	Original Author(s): Rob Remillard of Sodecia GTAC.; 
------------------------------------------------------------------------------------------
REVISION NOTES:
	Version 20150203
		- intial concept, r.remillard
	Version 20151105
		- added discrete_image to var_output to expose for visualization on UIs, b.lekx-toniolo
		- added Not Comm_Error interlock to Locked and Unlocked Signals for redundancy, b.lekx-toniolo
------------------------------------------------------------------------------------------
*)



FUNCTION_BLOCK FB_ATI_Changer_20151105

VAR_INPUT

	ATI_Lock_Requested:				BOOL;
	ATI_Unlock_Requested:			BOOL;
	Fault_Reset:						BOOL;

END_VAR

VAR

	In_From_Hardware AT %I*: 			udt_ATI_Input_20150203;
	Out_To_Hardware AT %Q*:			udt_ATI_Output_20150203;

	Lock_ATI:						BOOL;
	Unlock_ATI:						BOOL;

	(*Input Signals From ATI*)
	US1_Power_Present:				BOOL;
	US2_Power_Present:				BOOL;
	RTL1:							BOOL;
	RTL2:							BOOL;
	Tool_Present:					BOOL;
	Tool_PWR_Present:				BOOL;

	TSIV:							BOOL;
	TSRV:							BOOL;
	RTLV1:							BOOL;
	RTLV2:							BOOL;

	Tool_ID:							UDINT;

	Error_On_Lock:					BOOL;
	Error_On_Unlock:					BOOL;


	DiscreteNode_OK: 				BOOL;
	ECatSlave_Cable_Breaks:			UDINT;

END_VAR

VAR_OUTPUT

	FB_OK:							BOOL;
	Discrete_Image:					udt_ATIxx_Image_20151104;
	ATI_Sensors_On:					BOOL;
	ATI_Locked:						BOOL;
	ATI_Unlocked:					BOOL;
	ATI_Unlock_Enabled:				BOOL;
	Tool_ID_Out0:					BOOL;
	Tool_ID_Out1:					BOOL;
	Tool_ID_Out2:					BOOL;
	Tool_ID_Out3:					BOOL;
	Tool_ID_Out4:					BOOL;
	Tool_ID_Out5:					BOOL;
	Tool_ID_Out6:					BOOL;
	Tool_ID_Out7:					BOOL;
	Unsafe_Unlock:					BOOL;
	Sensor_Fault:						BOOL;
	COMM_Error:						BOOL;

END_VAR

	(*Set FB_OK to True*)
	FB_OK:= TRUE;

(*$$$$$$$$$$$$$$$$$$$$$$$$$$$$$$$$$$$$$$$$$$$$$$$$Gather Status Of Hardware $$$$$$$$$$$$$$$$$$$$$$$$$$$$$$$$$$$$$$$$$$$$$$$$$$$$*)
	(*Discrete I/O Nodes*)
	IF In_From_Hardware.InfoData.State=8

		THEN
			DiscreteNode_OK:=TRUE;

	ELSE
			DiscreteNode_OK:=FALSE;

	END_IF;


	(*Cable Break Detection*)
	ECatSlave_Cable_Breaks:= FUN_GTAC_EcatSlaveConnState
							(In_From_Hardware.InfoData.State,
							0,0,0,0,0,0,0,0,0,0,0,0,0,0,0,0,0,0,0,0,0,0,0,0,0,0,0,0,0); (*Function Returns Flags to warn of possible cable break*)

(*----------------------------------------------------------------------------------------------------------------------------------------------------------------------------------------------------------*)

(*+++++++++++++++++++++++++++Input Byte Mapping+++++++++++++++++++++++++++*)

	ATI_Locked:= In_From_Hardware.Byte0.0 AND NOT Comm_Error;				(*ATI Locked Status from VL1*)
	ATI_Unlocked:= In_From_Hardware.Byte0.1 AND NOT Comm_Error;				(*ATI Unlocked Status from VL1*)
	US1_Power_Present:= In_From_Hardware.Byte0.2;								(*ATI Main Power Present*)
	US2_Power_Present:= In_From_Hardware.Byte0.3;								(*ATI Valve Power Present*)
	RTL1:= In_From_Hardware.Byte0.4;											(*ATI Ready To Lock Prox 1*)
	RTL2:= In_From_Hardware.Byte0.5;											(*ATI Ready To Lock Prox 2*)
	Tool_Present:= In_From_Hardware.Byte0.6;									(*ATI Master and Tool are in Electrical Contact*)
	Tool_PWR_Present:= In_From_Hardware.Byte0.7;								(*ATI Arc Prevention Circuit on and power to Tool*)

	ATI_Unlock_Enabled:= In_From_Hardware.Byte1.0;								(*ATI Unlock Enabled*)
	TSIV:= In_From_Hardware.Byte1.1;											(*ATI Tool Stand Interlock Switch Verify*)
	TSRV:= In_From_Hardware.Byte1.2;											(*ATI Tool Stand Interlock Relay Verify*)
	RTLV1:= In_From_Hardware.Byte1.4;											(*ATI Ready To Lock Relay1 Verify*)
	RTLV2:= In_From_Hardware.Byte1.5;											(*ATI Ready To Lock Relay2 Verify*)

	Error_On_Lock:= In_From_Hardware.Byte2.0;									(*ATI Overload or Short Circuit on Latch Output*)
	Error_On_Unlock:= In_From_Hardware.Byte2.1;									(*ATI Overload or Short Circuit on Unlatch Output*)
	Unsafe_Unlock:= In_From_Hardware.Byte2.3;									(*ATI Unlatch rejected due to unsafe condition present*)
	Sensor_Fault:= In_From_Hardware.Byte2.4;									(*ATI Lock and Unlock inputs true at the same time*)
	COMM_Error:= In_From_Hardware.Byte2.5;									(*ATI Tool ID Communication Timeout*)

	Tool_ID:=  In_From_Hardware.Byte456;										(*ATI Tool ID*)

	Tool_ID_Out0:= Tool_ID.0;
	Tool_ID_Out1:= Tool_ID.1;
	Tool_ID_Out2:= Tool_ID.2;
	Tool_ID_Out3:= Tool_ID.3;
	Tool_ID_Out4:= Tool_ID.4;
	Tool_ID_Out5:= Tool_ID.5;
	Tool_ID_Out6:= Tool_ID.6;
	Tool_ID_Out7:= Tool_ID.7;



(*+++++++++++++++++++++++++++++ATI Control Code++++++++++++++++++++++++++++*)

	IF ATI_Lock_Requested
		THEN
			Lock_ATI:= TRUE;
			Unlock_ATI:= FALSE;
	ELSIF NOT Tool_Present AND NOT ATI_Lock_Requested
		THEN
			Lock_ATI:= FALSE;
	END_IF;

	IF ATI_Unlock_Requested AND TSIV AND TSRV AND ATI_Unlock_Enabled
		THEN
			Lock_ATI:= FALSE;
			Unlock_ATI:= NOT Lock_ATI;
	END_IF;

	ATI_Sensors_On:= RTL1 AND RTL2;

(*$$$$$$$$$$$$$$$$$$$$$$$$$$$$$$$$$$$$$$$$$$$$$$ Transfer Standard Outputs $$$$$$$$$$$$$$$$$$$$$$$$$$$$$$$$$$$$$$$$$$$*)
	(*Transfer I/O Images for Display On UI*)
Discrete_Image.In_From_Hardware:= In_From_Hardware;
Discrete_Image.Out_To_Hardware:= Out_To_Hardware;
Discrete_Image.ECatSlave_Cable_Breaks:= ECatSlave_Cable_Breaks;

(*+++++++++++++++++++++++++++Output Byte Mapping+++++++++++++++++++++++++++*)

	Out_To_Hardware.Byte0.0:= Lock_ATI;					(*Request Lock*)
	Out_To_Hardware.Byte0.1:= Unlock_ATI;					(*Request Unlock*)
	Out_To_Hardware.Byte0.3:= Fault_Reset;					(*Reset Errors, allow affected I/O to be reactivated*)

END_FUNCTION_BLOCK

// ---- POUs/FBs/FB_GTAC_WaterStand_20220622.TcPOU
(*FB to handle robot water tower
	Version: 20170801
	- combined FB_GTAC_Robot_TempFlow and FB_GTAC_Fixture_Single into one FB, j.vandongen
	- added option to choose between 1 output and 2 output (in the case of a fixture where only one is required), j.vandongen
	Version 20171111
	- changed Timeout reset to rising edge trigger, j.vandongen 
	- added var out for coolig ok, j.vandongen
	Version 20190726
	- added outputs for the control of the water saver unit, j.vandongen
	Version 20200710
	- removed cards EP3174 and EP2028. changed to EP6224 IO-Link, j.vandongen
	Version 20200917
	- corrected error in fault code for DegreesC2, j.vandongen
	Version 20201125
	- corrected mapping issue causing incorrect flow to be shown, j.vandongen
	Version 20220131
	- added mapping for using the inport ports in the I/O Link cards, j. underhill
	Version 20220622
	- fixes for issues found with negative flow values (see 5.06 GH issues #2 notes), b.lekx-toniolo, j.underhill, d.esteves, c.drees
		NOTE: (from brent) the issue is we take a signed value from the meter and shove it into a UINT bit by bit....I'm not sure why the original developer did this but it should be re-examined as a whole


*)

FUNCTION_BLOCK FB_GTAC_WaterStand_20220622

VAR_INPUT

	Enable_Timeout: BOOL; 	(*Enable Timeout to shut off valve if flow not achieved in time*)
	Timeout_Reset: BOOL;		(*Reset (Retry) Timepout*)
	Timeout_SetPoint: TIME;	(*TimeoutSetpoint Input, limited to 1-10S*)

	TempHighLimit1: REAL;
	TempHighLimit2: REAL;
	FlowLowLimit1: REAL;
	FlowLowLimit2: REAL;

	Option_WaterCount: INT;

	Valve1: BOOL;
	Valve2: BOOL;
	Valve3: BOOL;
	Valve4: BOOL;


END_VAR

VAR

(*Hardware Related Data Types*)
	(*Develop "Beckhoff Nodes"*)
	N01 AT %I*: udt_EP6224;
	N01_I AT %I*: udt_EP6224_I;
	N01_CMD AT %Q*: udt_EP6224_CMD;

(* Nodes States*)
	DiscreteNode_OK: BOOL;

(*Cable Break States*)
	ECatSlave_Cable_Breaks: UDINT;

	Fault_Tmrs: ARRAY [0..10] OF TON;
	Temperature1_Fault_Delay_TMR : BOOL;
	Temperature2_Fault_Delay_TMR : BOOL;
	Flow1_Fault_Delay_TMR : BOOL;
	Flow2_Fault_Delay_TMR : BOOL;

	RawTemp1: UINT;
	RawTemp2: UINT;

	RawFlow1: UINT;
	RawFlow2: UINT;

	TempReal1: REAL;
	TempReal2: REAL;
	FlowReal1: REAL;
	FlowReal2: REAL;

	DegreesC1: REAL;
	DegreesC2: REAL;

	Flow_lpm1: REAL;
	Flow_lpm2: REAL;

	WaterTempFlow_OK: BOOL;

	Reset_Req: R_TRIG;


END_VAR

VAR_OUTPUT

	Discrete_Image: udt_WaterStand_Image_20220131;

	Temperature_Fault1: BOOL;
	Temperature_Fault2: BOOL;
	Flow_Fault1: BOOL;
	Flow_Fault2: BOOL;

	Cooling_OK: BOOL;

END_VAR

(*$$$$$$$$$$$$$$$$$$$$$$$$$$$$$$$$$$$$$$$$$$$$$$$$Gather Status Of Hardware $$$$$$$$$$$$$$$$$$$$$$$$$$$$$$$$$$$$$$$$$$$$$$$$$$$$*)
	(*Discrete I/O Nodes*)
	IF (N01.InfoData.State=8)

		THEN DiscreteNode_OK:=TRUE;
	ELSE DiscreteNode_OK:=FALSE;
	END_IF;
	(*Cable Break Detection*)
	ECatSlave_Cable_Breaks:= FUN_GTAC_EcatSlaveConnState
							(N01.InfoData.State,
							0,0,0,0,0,0,0,0,0,0,0,0,0,0,0,0,0,0,0,0,0,0,0,0,0,0,0,0,0); (*Function Returns Flags to warn of possible cable break*)




(*----------------------------------------------------Temperature conversion and output----------------------------------------------------*)
	RawTemp1.0:= N01.Port1_ProcessData[7].2;
	RawTemp1.1:= N01.Port1_ProcessData[7].3;
	RawTemp1.2:= N01.Port1_ProcessData[7].4;
	RawTemp1.3:= N01.Port1_ProcessData[7].5;
	RawTemp1.4:= N01.Port1_ProcessData[7].6;
	RawTemp1.5:= N01.Port1_ProcessData[7].7;
	RawTemp1.6:= N01.Port1_ProcessData[6].0;
	RawTemp1.7:= N01.Port1_ProcessData[6].1;
	RawTemp1.8:= N01.Port1_ProcessData[6].2;
	RawTemp1.9:= N01.Port1_ProcessData[6].3;
	RawTemp1.10:= N01.Port1_ProcessData[6].4;
	RawTemp1.11:= N01.Port1_ProcessData[6].5;
	RawTemp1.12:= N01.Port1_ProcessData[6].6;
	RawTemp1.13:= N01.Port1_ProcessData[6].7;

	TempReal1:= RawTemp1 * 0.1; (*gradient to shift decimal place*)

	RawTemp2.0:= N01.Port2_ProcessData[7].2;
	RawTemp2.1:= N01.Port2_ProcessData[7].3;
	RawTemp2.2:= N01.Port2_ProcessData[7].4;
	RawTemp2.3:= N01.Port2_ProcessData[7].5;
	RawTemp2.4:= N01.Port2_ProcessData[7].6;
	RawTemp2.5:= N01.Port2_ProcessData[7].7;
	RawTemp2.6:= N01.Port2_ProcessData[6].0;
	RawTemp2.7:= N01.Port2_ProcessData[6].1;
	RawTemp2.8:= N01.Port2_ProcessData[6].2;
	RawTemp2.9:= N01.Port2_ProcessData[6].3;
	RawTemp2.10:= N01.Port2_ProcessData[6].4;
	RawTemp2.11:= N01.Port2_ProcessData[6].5;
	RawTemp2.12:= N01.Port2_ProcessData[6].6;
	RawTemp2.13:= N01.Port2_ProcessData[6].7;

	TempReal2:= RawTemp2 * 0.1; (*gradient to shift decimal place*)

(*Set the scale of the input value to match the temperature switch*)
	DegreesC1:= TempReal1;			(*Scale value determined at setup*)
	DegreesC2:= TempReal2;			(*Scale value determined at setup*)



(*----------------------------------------------------------Flow conversion and Output-------------------------------------------------------*)
	RawFlow1.0:= N01.Port1_ProcessData[5].0;
	RawFlow1.1:= N01.Port1_ProcessData[5].1;
	RawFlow1.2:= N01.Port1_ProcessData[5].2;
	RawFlow1.3:= N01.Port1_ProcessData[5].3;
	RawFlow1.4:= N01.Port1_ProcessData[5].4;
	RawFlow1.5:= N01.Port1_ProcessData[5].5;
	RawFlow1.6:= N01.Port1_ProcessData[5].6;
	RawFlow1.7:= N01.Port1_ProcessData[5].7;
	RawFlow1.8:= N01.Port1_ProcessData[4].0;
	RawFlow1.9:= N01.Port1_ProcessData[4].1;
	RawFlow1.10:= N01.Port1_ProcessData[4].2;
	RawFlow1.11:= N01.Port1_ProcessData[4].3;
	RawFlow1.12:= N01.Port1_ProcessData[4].4;
	RawFlow1.13:= N01.Port1_ProcessData[4].5;
	RawFlow1.14:= N01.Port1_ProcessData[4].6;
	(*RawFlow1.15:= N01.Port1_ProcessData[4].7;*)

IF N01.Port1_ProcessData[4].7		(*Bool that indicates the negative part of the word DE*)
	THEN
	FlowReal1:= 0; (*gradient to shift decimal place*)
ELSE
	FlowReal1:= RawFlow1 * 0.01; (*gradient to shift decimal place*)
END_IF

	RawFlow2.0:=  N01.Port2_ProcessData[5].0;
	RawFlow2.1:=  N01.Port2_ProcessData[5].1;
	RawFlow2.2:=  N01.Port2_ProcessData[5].2;
	RawFlow2.3:=  N01.Port2_ProcessData[5].3;
	RawFlow2.4:=  N01.Port2_ProcessData[5].4;
	RawFlow2.5:=  N01.Port2_ProcessData[5].5;
	RawFlow2.6:=  N01.Port2_ProcessData[5].6;
	RawFlow2.7:=  N01.Port2_ProcessData[5].7;
	RawFlow2.8:=  N01.Port2_ProcessData[4].0;
	RawFlow2.9:=  N01.Port2_ProcessData[4].1;
	RawFlow2.10:= N01.Port2_ProcessData[4].2;
	RawFlow2.11:= N01.Port2_ProcessData[4].3;
	RawFlow2.12:= N01.Port2_ProcessData[4].4;
	RawFlow2.13:= N01.Port2_ProcessData[4].5;
	RawFlow2.14:= N01.Port2_ProcessData[4].6;
	(*RawFlow2.15:= N01.Port2_ProcessData[4].7;*)

IF N01.Port2_ProcessData[4].7		(*Bool that indicates the negative part of the word DE*)
	THEN
	FlowReal2:= 0; (*gradient to shift decimal place*)
ELSE
	FlowReal2:= RawFlow2 * 0.01; (*gradient to shift decimal place*)
END_IF

(*Set the scale of the input value to match the flow switch*)
	Flow_lpm1:= FlowReal1;			(*Scale value determined at setup*)
	Flow_lpm2:= FlowReal2;			(*Scale value determined at Setup*)

(*Bottom at zero if flow values go negative as we're only interested in one direction of flow*)
IF (Flow_lpm1 < 0)
	THEN
	Flow_lpm1:= 0;
END_IF

IF (Flow_lpm2 < 0)
	THEN
	Flow_lpm2:= 0;
END_IF

(*-------------------------------------------------------Temperature and Flow Fault Status--------------------------------------------------*)
(*Determine if there is a Temperature fault*)

(*Temperature1 Fault Delay Timer*)
	Fault_Tmrs[1].PT:= T#2.0s;
	Fault_Tmrs[1]();
	Fault_Tmrs[1].IN:= (DegreesC1 > TempHighLimit1) OR (DegreesC1 < 2);
	Temperature1_Fault_Delay_TMR :=Fault_Tmrs[1].Q;
	Temperature_Fault1:=  ((DegreesC1 > TempHighLimit1) OR (DegreesC1 < 2)) AND Temperature1_Fault_Delay_TMR;

(*Temperature2 Fault Delay Timer*)
	Fault_Tmrs[2].PT:= T#2.0s;
	Fault_Tmrs[2]();
	Fault_Tmrs[2].IN:= (DegreesC2 > TempHighLimit2) OR (DegreesC2 < 2);
	Temperature2_Fault_Delay_TMR :=Fault_Tmrs[2].Q;
	Temperature_Fault2:= ((DegreesC2> TempHighLimit2) OR (DegreesC2 < 2)) AND Temperature2_Fault_Delay_TMR;


(*-------------------- Determine if there is a flow fault --------------------------*)

(*Place Boundries on Flow Setpoint Timeout input*)
	IF (Timeout_SetPoint <T#1.0s) OR (Timeout_SetPoint >T#10.0S)
		THEN
		Timeout_SetPoint:= T#5.0s;
	END_IF;

	Reset_Req(
			CLK:= Timeout_Reset,
			Q=>
			);


(*Flow1 Fault Delay Timer*)
	Fault_Tmrs[3].PT:= Timeout_Setpoint;
	Fault_Tmrs[3]();
	Fault_Tmrs[3].IN:= Flow_lpm1 < FlowLowLimit1 AND NOT Reset_Req.Q AND Valve1;
	Flow1_Fault_Delay_TMR :=Fault_Tmrs[3].Q;

	IF (Flow_lpm1 < FlowLowLimit1) AND Flow1_Fault_Delay_TMR
		THEN
			Flow_Fault1:= TRUE;
		ELSE
			Flow_Fault1:= FALSE;
	END_IF;

(*Flow2 Fault Delay Timer*)
	Fault_Tmrs[4].PT:= Timeout_Setpoint;
	Fault_Tmrs[4]();
	Fault_Tmrs[4].IN:= (Flow_lpm2 < FlowLowLimit2) AND NOT Reset_Req.Q AND Valve1;
	Flow2_Fault_Delay_TMR :=Fault_Tmrs[4].Q;

	IF (Flow_lpm2 < FlowLowLimit2) AND Flow2_Fault_Delay_TMR
		THEN
			Flow_Fault2:= TRUE;
		ELSE
			Flow_Fault2:= FALSE;
	END_IF;


(*----------------------------------Transfer Data to Discrete Image------------------*)
	Discrete_Image.N01:= N01;
	Discrete_Image.N01_CMD:= N01_CMD;
	Discrete_Image.Water_Flow_Gun:= Flow_Lpm1;
	Discrete_Image.Water_Flow_Trans:= Flow_Lpm2;
	Discrete_Image.Water_Temp_Gun:= DegreesC1;
	Discrete_Image.Water_Temp_Trans:= DegreesC2;
	Discrete_Image.ECatSlave_Cable_Breaks:= EcatSlave_Cable_Breaks;


(*----------------------------------------Output Final State-----------------------------------------*)
	WaterTempFlow_OK:= NOT Flow_Fault1 AND NOT Temperature_Fault1 AND ((NOT Flow_Fault2  AND NOT Temperature_Fault2) OR (Option_WaterCount=1));

	Cooling_OK:= WaterTempFlow_OK AND Valve1
			AND (Flow_lpm1 > FlowLowLimit1)
			AND ((Flow_lpm2 > FlowLowLimit2) OR (Option_WaterCount=1));



(*-----------------------------------------------------------------Valve Control-------------------------------------------------------------------*)
(*Control the valve*)
	N01_CMD.Port3_Q:= Valve1 AND NOT (( Flow_Fault1 OR  Flow_Fault2) AND Enable_Timeout);



(*end*)

END_FUNCTION_BLOCK

// ---- POUs/FUNs/FUN_GTAC_GenericRobotInputImage_From_KUKAKRC4.TcPOU
(*Function used during SIM to map KUKA FB Bit Typed Output Data to HW Byte Array Typed Image, simply for UI display
	author: Brent Lekx-Toniolo of Sodecia GTAC
	date: January 2024

	Last Edit: Jan 22, 2024, BLT
*)

FUNCTION FUN_GTAC_GenericRobotInputImage_From_KUKAKRC4 : udt_GenericRobot_AnyFieldbus_InputBytes_20220421
VAR_INPUT
	BitBased_Data: udt_EtherCAT_Kuka_InputBits_20121204;


END_VAR
VAR
	Bit_Index: INT;
	Byte_Index: INT;
	BytesBit_Index: BYTE;
END_VAR

(*Ensure Index is reset*)
Bit_Index:= 1;
(*Gathering of Robot Specific Data Type Points to Map to Generic Byte Typed Array*)
FOR Byte_Index:=1 TO 64 BY 1 DO
			FUN_GTAC_GenericRobotInputImage_From_KUKAKRC4.Byte_[Byte_Index].0:= BitBased_Data.Robot_OUT[Bit_Index];
			Bit_Index:=Bit_Index+1;
			FUN_GTAC_GenericRobotInputImage_From_KUKAKRC4.Byte_[Byte_Index].1:= BitBased_Data.Robot_OUT[Bit_Index];
			Bit_Index:=Bit_Index+1;
			FUN_GTAC_GenericRobotInputImage_From_KUKAKRC4.Byte_[Byte_Index].2:= BitBased_Data.Robot_OUT[Bit_Index];
			Bit_Index:=Bit_Index+1;
			FUN_GTAC_GenericRobotInputImage_From_KUKAKRC4.Byte_[Byte_Index].3:= BitBased_Data.Robot_OUT[Bit_Index];
			Bit_Index:=Bit_Index+1;
			FUN_GTAC_GenericRobotInputImage_From_KUKAKRC4.Byte_[Byte_Index].4:= BitBased_Data.Robot_OUT[Bit_Index];
			Bit_Index:=Bit_Index+1;
			FUN_GTAC_GenericRobotInputImage_From_KUKAKRC4.Byte_[Byte_Index].5:= BitBased_Data.Robot_OUT[Bit_Index];
			Bit_Index:=Bit_Index+1;
			FUN_GTAC_GenericRobotInputImage_From_KUKAKRC4.Byte_[Byte_Index].6:= BitBased_Data.Robot_OUT[Bit_Index];
			Bit_Index:=Bit_Index+1;
			FUN_GTAC_GenericRobotInputImage_From_KUKAKRC4.Byte_[Byte_Index].7:= BitBased_Data.Robot_OUT[Bit_Index];
			Bit_Index:=Bit_Index+1;
	END_FOR;

END_FUNCTION

// ---- POUs/FUNs/FUN_GTAC_GenericRobotInputImage_TO_KUKAKRC4.TcPOU
(*Function used to map HW Byte Array Typed Generic Input Image (from Robot Outputs) to KUKA FB Bit Typed Data
to more closly ressemble Robot Output structure in teach pendant
	author: Brent Lekx-Toniolo of Sodecia GTAC
	date: November 2012
	version 1.0
		- initial concept

	Last Edit: December 4th, 2012, BLT

*)

FUNCTION FUN_GTAC_GenericRobotInputImage_TO_KUKAKRC4 : udt_EtherCAT_Kuka_InputBits_20121204
VAR_INPUT
	ByteBased_Array: udt_GenericRobot_AnyFieldbus_InputBytes_20220421;


END_VAR
VAR
	Bit_Index: INT;
	Byte_Index: INT;
	BytesBit_Index: BYTE;
END_VAR

(*Ensure Index is reset*)
Bit_Index:= 1;
(*Gathering of Generic Byte Typed Array to map to Robot Specific Data Type Points*)
	FOR Byte_Index:=1 TO 64 BY 1 DO
			FUN_GTAC_GenericRobotInputImage_TO_KUKAKRC4.Robot_OUT[Bit_Index]:= ByteBased_Array.Byte_[Byte_Index].0;
			Bit_Index:=Bit_Index+1;
			FUN_GTAC_GenericRobotInputImage_TO_KUKAKRC4.Robot_OUT[Bit_Index]:= ByteBased_Array.BYTE_[Byte_Index].1;
			Bit_Index:=Bit_Index+1;
			FUN_GTAC_GenericRobotInputImage_TO_KUKAKRC4.Robot_OUT[Bit_Index]:= ByteBased_Array.BYTE_[Byte_Index].2;
			Bit_Index:=Bit_Index+1;
			FUN_GTAC_GenericRobotInputImage_TO_KUKAKRC4.Robot_OUT[Bit_Index]:= ByteBased_Array.BYTE_[Byte_Index].3;
			Bit_Index:=Bit_Index+1;
			FUN_GTAC_GenericRobotInputImage_TO_KUKAKRC4.Robot_OUT[Bit_Index]:= ByteBased_Array.BYTE_[Byte_Index].4;
			Bit_Index:=Bit_Index+1;
			FUN_GTAC_GenericRobotInputImage_TO_KUKAKRC4.Robot_OUT[Bit_Index]:= ByteBased_Array.BYTE_[Byte_Index].5;
			Bit_Index:=Bit_Index+1;
			FUN_GTAC_GenericRobotInputImage_TO_KUKAKRC4.Robot_OUT[Bit_Index]:= ByteBased_Array.BYTE_[Byte_Index].6;
			Bit_Index:=Bit_Index+1;
			FUN_GTAC_GenericRobotInputImage_TO_KUKAKRC4.Robot_OUT[Bit_Index]:= ByteBased_Array.BYTE_[Byte_Index].7;
			Bit_Index:=Bit_Index+1;
	END_FOR;

END_FUNCTION

// ---- POUs/FUNs/FUN_GTAC_KUKAKRC4_To_GenericRobotOutputImage.TcPOU
(*Function used to map KUKA FB Bit Typed Data to HW Byte Array Typed Generic Output Image (to Robot Inputs)
to more closly ressemble Robot Input structure in teach pendant
	author: Brent Lekx-Toniolo of Sodecia GTAC
	date: November 2012
	version 1.0
		- initial concept


	Last Edit: December 4th, 2012, BLT
*)

FUNCTION FUN_GTAC_KUKAKRC4_To_GenericRobotOutputImage : udt_GenericRobot_AnyFieldbus_OutputBytes_20220421
VAR_INPUT
	BitBased_Data: udt_EtherCAT_Kuka_OutputBits_20121204;


END_VAR
VAR
	Bit_Index: INT;
	Byte_Index: INT;
	BytesBit_Index: BYTE;
END_VAR

(*Ensure Index is reset*)
Bit_Index:= 1;
(*Gathering of Robot Specific Data Type Points to Map to Generic Byte Typed Array*)
FOR Byte_Index:=1 TO 64 BY 1 DO
			FUN_GTAC_KUKAKRC4_To_GenericRobotOutputImage.Byte_[Byte_Index].0:= BitBased_Data.Robot_IN[Bit_Index];
			Bit_Index:=Bit_Index+1;
			FUN_GTAC_KUKAKRC4_To_GenericRobotOutputImage.Byte_[Byte_Index].1:= BitBased_Data.Robot_IN[Bit_Index];
			Bit_Index:=Bit_Index+1;
			FUN_GTAC_KUKAKRC4_To_GenericRobotOutputImage.Byte_[Byte_Index].2:= BitBased_Data.Robot_IN[Bit_Index];
			Bit_Index:=Bit_Index+1;
			FUN_GTAC_KUKAKRC4_To_GenericRobotOutputImage.Byte_[Byte_Index].3:= BitBased_Data.Robot_IN[Bit_Index];
			Bit_Index:=Bit_Index+1;
			FUN_GTAC_KUKAKRC4_To_GenericRobotOutputImage.Byte_[Byte_Index].4:= BitBased_Data.Robot_IN[Bit_Index];
			Bit_Index:=Bit_Index+1;
			FUN_GTAC_KUKAKRC4_To_GenericRobotOutputImage.Byte_[Byte_Index].5:= BitBased_Data.Robot_IN[Bit_Index];
			Bit_Index:=Bit_Index+1;
			FUN_GTAC_KUKAKRC4_To_GenericRobotOutputImage.Byte_[Byte_Index].6:= BitBased_Data.Robot_IN[Bit_Index];
			Bit_Index:=Bit_Index+1;
			FUN_GTAC_KUKAKRC4_To_GenericRobotOutputImage.Byte_[Byte_Index].7:= BitBased_Data.Robot_IN[Bit_Index];
			Bit_Index:=Bit_Index+1;
	END_FOR;

END_FUNCTION

// ---- POUs/FUNs/FUN_GTAC_DEGtoINDEX.TcPOU
(*
Function to dirve Robot Animation Symbol on UI,
	- Two Inputs are exposed to the programmer:
		- i_Raw_Degrees (Int), this is a 0-360 degree value sent from the Robot S-Axis
		- i_Home_Offset (Int), a stsic value set by a Robot FB Input to orient the Animations "Zero position" to match the physical instal position of the robot with resepct to 12 o'clock

	author(s): Brent Lekx-Toniolo and JVD OF Sodecia GTAC
	UI Symbol author(s): Chris TImmermans of Edge Automation
	DATE: November 2014
	version 1.0
		- initial concept


	Last Edit: November, 2014, BLT
*)

FUNCTION FUN_GTAC_DEGtoINDEX : INT
VAR_INPUT
	i_Raw_Degrees: INT;
	i_Home_Offset: INT;		(*To Re-Orient the Robot from -180 to +180 degrees*)

END_VAR
VAR
	i_Raw_Degrees_Bound: INT;
	i_Homed_Degrees: INT;
END_VAR

(*Develop Homed Position based on raw data plus install offset*)

IF (i_Raw_Degrees >=0) AND (i_Raw_Degrees<=360) (*Do Bound Checking on Raw Position*)
	THEN
	i_Raw_Degrees_Bound:= i_Raw_Degrees;
ELSIF (i_Raw_Degrees >360)
	THEN
	i_Raw_Degrees_Bound:= 360;
ELSIF (i_Raw_Degrees <0)
	THEN
	i_Raw_Degrees_Bound:= 0;
END_IF;



	IF (i_Home_Offset >=0) AND (i_Home_Offset<360) (*Do Bound Checking on Offset Position*)
		THEN
		IF ((i_Raw_Degrees_Bound+i_Home_Offset-186)>=0) AND ((i_Raw_Degrees_Bound+i_Home_Offset-186)<=360) (*If Raw Data from Robot + Home Offset value reachs bounds of 0 or 360, then wrap around*)
			THEN
				i_Homed_Degrees:= i_Raw_Degrees_Bound+i_Home_Offset-186;
		ELSIF ((i_Raw_Degrees_Bound+i_Home_Offset)>186)
			THEN
				i_Homed_Degrees:= ((i_Raw_Degrees_Bound+i_Home_Offset-186)-360);
		ELSIF ((i_Raw_Degrees_Bound+i_Home_Offset)<=186)
			THEN
				i_Homed_Degrees:= 360-((360-(i_Raw_Degrees_Bound+i_Home_Offset-186))-360);
		END_IF;
	END_IF;

(*Set 10 Degree Slices as bounds for Indexing trigger points to UI Images*)
FUN_GTAC_DEGtoINDEX:= (i_Homed_Degrees/10)*10;

END_FUNCTION

// ---- POUs/FUNs/FUN_GTAC_BOOLStoINT.TcPOU
(*Copy Individual BOOLS (input to the FUN), into individual bits of the INT Return
	author: Brent Lekx-Toniolo OF Sodecia GTAC
	date: November 2012
	version 1.0
		- initial concept


	Last Edit: December 3rd, 2012, BLT
*)

FUNCTION FUN_GTAC_BOOLStoINT : INT
VAR_INPUT
	Bool0: BOOL;
	Bool1: BOOL;
	Bool2: BOOL;
	Bool3: BOOL;
	Bool4: BOOL;
	Bool5: BOOL;
	Bool6: BOOL;
	Bool7: BOOL;
	Bool8: BOOL;
	Bool9: BOOL;
	Bool10: BOOL;
	Bool11: BOOL;
	Bool12: BOOL;
	Bool13: BOOL;
	Bool14: BOOL;
	Bool15: BOOL;
END_VAR
VAR
END_VAR

(*Copy Individual BOOLS (input to the FUN) into individual bits of the INT Return*)

FUN_GTAC_BOOLStoINT.0:= Bool0;
FUN_GTAC_BOOLStoINT.1:= Bool1;
FUN_GTAC_BOOLStoINT.2:= Bool2;
FUN_GTAC_BOOLStoINT.3:= Bool3;
FUN_GTAC_BOOLStoINT.4:= Bool4;
FUN_GTAC_BOOLStoINT.5:= Bool5;
FUN_GTAC_BOOLStoINT.6:= Bool6;
FUN_GTAC_BOOLStoINT.7:= Bool7;
FUN_GTAC_BOOLStoINT.8:= Bool8;
FUN_GTAC_BOOLStoINT.9:= Bool9;
FUN_GTAC_BOOLStoINT.10:= Bool10;
FUN_GTAC_BOOLStoINT.11:= Bool11;
FUN_GTAC_BOOLStoINT.12:= Bool12;
FUN_GTAC_BOOLStoINT.13:= Bool13;
FUN_GTAC_BOOLStoINT.14:= Bool14;
FUN_GTAC_BOOLStoINT.15:= Bool15;

END_FUNCTION

// ---- POUs/FBs/FB_GTAC_SS_20250407.TcPOU
(*FB used to Handle Large Service Stand I/O

------------------------------------------------------------------------
REVISION NOTES:
	Original Author(s): b.lekx-toniolo of Sodecia GTAC (broken out from Original grouped FB created by r.remillard); 
	Version 2015
		- Broke out from originally grouped "WS" FB, b.lekx-toniolo
	Version 20151209
		- Added changes for redundant valves, b.lekx-toniolo
	Version 20160713
		- Modified I/O structure to clean things up with redudant valve, b.lekx-toniolo
		- Added EDM_Fault to check for improper redundant valve action, b.lekx-toniolo
	Version 20171031
		-Added external control of outputs, j.vandongen
	Version 20250704
		-Adding in EP9218, r.jones
------------------------------------------------------------------------
*)


FUNCTION_BLOCK FB_GTAC_SS_20250407

VAR_INPUT

	Prev_EcatNode_Present: BOOL;
	Output_REQ: UDINT;
	Option_EP9214_Count: INT;
	FB_In: udt_Generic_EP9214_20250714;

END_VAR

VAR

	N01 AT %I*: udt_EP9128_20250704;
	N02 AT %I*: udt_EP1008_002_v2;
	N03 AT %Q*: udt_EP2028_002_v2;
	N03_STAT AT %I*: udt_EP2028_002_STAT;
	N04_STAT AT %I*: udt_EP9214_STAT_20250704;
	N04_CMD AT %Q*: udt_EP9214_CMD_20250704;
	(*Optional Power Distribution Blocks*)
	N999_STAT AT %I*: udt_EP9214_STAT_20250704;
	N999_CMD AT %Q*: udt_EP9214_CMD_20250704;
	N1000_STAT AT %I*: udt_EP9214_STAT_20250704;
	N1000_CMD AT %Q*: udt_EP9214_CMD_20250704;
	N1001_STAT AT %I*: udt_EP9214_STAT_20250704;
	N1001_CMD AT %Q*: udt_EP9214_CMD_20250704;	


	(*Cable Break Warning Flags*)(*Node States*)
	DiscreteNode_OK: BOOL;
	EP2028_NotPresent: BOOL;
	EP2028_PortB_MissingLnk: BOOL;
	EP1008_NotPresent: BOOL;
	EP1008_PortB_MissingLink: BOOL;
	ECatSlave_Cable_Breaks: UDINT;
	EP9128_NotPresent :BOOL;				(*is Not Present*)
	EP9128_PortD_MissingLink: BOOL;			(*SectionD Link 1 is for X2*)
	EP9128_PortD_MissingLink2: BOOL;		(*SectionD Link 2 is for X3*)
	EP9128_PortD_MissingLink3: BOOL;		(*SectionD Link 3 is for X6*)
	EP9128_PortB_MissingLink: BOOL;			(*SectionB Link 1 is for X4*)
	EP9128_PortB_MissingLink2: BOOL;		(*SectionB Link 2 is for X5*)
	EP9128_PortB_MissingLink3: BOOL;		(*SectionB Link 2 is for X7*)
	EP9128_PortC_MissingLink: BOOL;			(*SectionC is for Second section of Internal Fixtures X8*)
	EP9214_NotPresent :BOOL;	
	EP9214_PortB_MissingLnk: BOOL;
	N999_Missing: BOOL;
	N1000_Missing:BOOL; 					(*Second EP9224 Missing*)
	N1001_Missing:BOOL;						(*Third EP9224 Missing*)

END_VAR

VAR_OUTPUT

	Air_PressureOK: BOOL;
	Valve1_Off: BOOL;
	Valve2_Off: BOOL;
	Valves_Off: BOOL;
	EDM_Fault: BOOL;
	Discrete_Image: udt_SSxx_Image_20250704;

END_VAR


(*$$$$$$$$$$$$$$$$$$$$$$$$$$$$$$$$$$$$$$$$$$$$$$$$Gather Status Of Hardware $$$$$$$$$$$$$$$$$$$$$$$$$$$$$$$$$$$$$$$$$$$$$$$$$$$$*)
	(*Discrete I/O Node*)
	IF (N01.InfoData.State=8) AND (N01.InfoDataB.State=8) AND (N01.InfoDataC.State=8) AND (N02.InfoData.State=8)
		AND (N03_STAT.InfoData.State=8) AND (N04_STAT.InfoData.State=8)
		AND ((N999_STAT.InfoData.State=8) OR FB_In.Option_EP9214_Count < 1)
		AND ((N1000_STAT.InfoData.State=8) OR FB_In.Option_EP9214_Count < 2)
		AND ((N1001_STAT.InfoData.State=8) OR FB_In.Option_EP9214_Count < 3)
		THEN DiscreteNode_OK:=TRUE;
	ELSE DiscreteNode_OK:=FALSE;
	END_IF;
	
	IF ((N01.InfoData.State=257) AND (N01.InfoDataB.State=257) AND (N01.InfoDataC.State=257))
		THEN EP9128_NotPresent:= TRUE;				(*Port X1*)
	ELSE EP9128_NotPresent:= FALSE;
	END_IF;	
	
	IF ((N01.InfoData.State=33800) OR (N01.InfoData.State=41992))
		THEN EP9128_PortD_MissingLink:= TRUE;		(*PortD Attached at Port X2*)
	ELSE EP9128_PortD_MissingLink:= FALSE;
	END_IF;

	IF  ((N01.InfoData.State=9224) OR (N01.InfoData.State=41992))
		THEN EP9128_PortB_MissingLink:= TRUE;		(*PortB Attached at Port X3*)
	ELSE EP9128_PortB_MissingLink:= FALSE;
	END_IF;

	IF ((N01.InfoDataB.State=33800) OR (N01.InfoDataB.State=41992))
		THEN EP9128_PortD_MissingLink2:= TRUE;		(*PortD Attached at Port X4*)
	ELSE EP9128_PortD_MissingLink2:= FALSE;
	END_IF;

	IF  ((N01.InfoDataB.State=9224) OR (N01.InfoDataB.State=41992))
		THEN EP9128_PortB_MissingLink2:= TRUE;		(*PortB Attached at Port X5*)
	ELSE EP9128_PortB_MissingLink2:= FALSE;
	END_IF;

	IF ((N01.InfoDataC.State=33800) OR (N01.InfoDataC.State=41992)
		OR (N01.InfoDataC.State=50184) OR (N01.InfoDataC.State=58376))
		THEN EP9128_PortD_MissingLink3:= TRUE;		(*PortD Attached at Port X6*)
	ELSE EP9128_PortD_MissingLink3:= FALSE;
	END_IF;

	IF  ((N01.InfoDataC.State=9224) OR (N01.InfoDataC.State=25608)
		OR (N01.InfoDataC.State=41992) OR (N01.InfoDataC.State=58376))
		THEN EP9128_PortB_MissingLink3:= TRUE;		(*PortB Attached at Port X7*)
	ELSE EP9128_PortB_MissingLink3:= FALSE;
	END_IF;

	IF  ((N01.InfoDataC.State=17416) OR (N01.InfoDataC.State=25608)
		OR (N01.InfoDataC.State=50184) OR (N01.InfoDataC.State=58376))
		THEN EP9128_PortC_MissingLink:= TRUE;		(*PortC Attached at Port X8*)
	ELSE EP9128_PortC_MissingLink:= FALSE;
	END_IF;
	
	IF N02.InfoData.State = 257 (*State Machine for Slave Not Present*)
		THEN EP1008_NotPresent:= TRUE;
	ELSE EP1008_NotPresent:= FALSE;
	END_IF;

	IF N03_STAT.InfoData.State = 257  (*State Machine for Slave Not Present*)
		THEN EP2028_NotPresent:= TRUE;
	ELSE EP2028_NotPresent:= FALSE;
	END_IF;

	IF N04_STAT.InfoData.State = 257  (*State Machine for Slave Not Present*)
		THEN EP9214_NotPresent:= TRUE;
	ELSE EP9214_NotPresent:= FALSE;
	END_IF;
	
	IF N04_STAT.InfoData.State = 9224  (*State Machine for Slave Not Present Port B*)
		THEN EP9214_PortB_MissingLnk:= TRUE;
	ELSE EP9214_PortB_MissingLnk:= FALSE;
	END_IF;
	
	IF (N999_Stat.InfoData.State=9224) AND (FB_In.Option_EP9214_Count >=1) (*State 9224 is missing link on port B*)
		THEN N999_Missing:= TRUE;
	ELSE N999_Missing := FALSE;
	END_IF;
	
	IF (N1000_Stat.InfoData.State=9224) AND (FB_In.Option_EP9214_Count >=2) (*State 9224 is missing link on port B*)
		THEN N1000_Missing:= TRUE;
	ELSE N1000_Missing := FALSE;
	END_IF;
	
	IF (N1001_Stat.InfoData.State=9224) AND (FB_In.Option_EP9214_Count >=3) (*State 9224 is missing link on port B*)
		THEN N1001_Missing:= TRUE;
	ELSE N1001_Missing := FALSE;
	END_IF;
	
	(*Wrap up break Flags to Variable for shipment to UI*)
	ECatSlave_Cable_Breaks.0:= EP9128_NotPresent AND Prev_EcatNode_Present;
	ECatSlave_Cable_Breaks.1:= EP1008_NotPresent AND NOT EP9128_NotPresent;
	ECatSlave_Cable_Breaks.2:= EP2028_NotPresent AND NOT EP1008_NotPresent;
	ECatSlave_Cable_Breaks.3:= EP9214_NotPresent AND NOT EP2028_NotPresent;
	ECatSlave_Cable_Breaks.4:= EP9214_PortB_MissingLnk;

	ECatSlave_Cable_Breaks.17:= EP9128_PortD_MissingLink; (*x2*)
	ECatSlave_Cable_Breaks.18:= EP9128_PortB_MissingLink; (*x3*)
	ECatSlave_Cable_Breaks.19:= EP9128_PortD_MissingLink2; (*x4*)
	ECatSlave_Cable_Breaks.20:= EP9128_PortB_MissingLink2; (*x5*)
	ECatSlave_Cable_Breaks.21:= EP9128_PortD_MissingLink3; (*x6*)
	ECatSlave_Cable_Breaks.22:= EP9128_PortB_MissingLink3; (*x7*)
	ECatSlave_Cable_Breaks.23:= EP9128_PortC_MissingLink; (*x8*)
	EcatSlave_Cable_Breaks.24:= N999_Missing;	
	EcatSlave_Cable_Breaks.25:= N1000_Missing;
	EcatSlave_Cable_Breaks.26:= N1001_Missing;

(*----------------------------------------------------- Map I/O---------------------------------------------*)

(*EP1008*)
Valve1_Off:= (*N02.I.0*) NOT N02.I.2;
Valve2_Off:= (*N02.I.1*) NOT N02.I.3;
Valves_Off:= Valve1_Off AND Valve2_Off;

Air_PressureOK:= (*N02.I.2*)N02.I.3;

(*EP2028*)
N03.Q.0:= Output_Req.0;			(*Enable Valve Sol.1*)
N03.Q.1:= Output_Req.1;			(*Enable Valve Sol.2*)
N03.Q.2:= Output_Req.2;
N03.Q.3:= Output_Req.3;
N03.Q.4:= Output_Req.4;
N03.Q.5:= Output_Req.5;
N03.Q.6:= Output_Req.6;
N03.Q.7:= Output_Req.7;


(*--------------------------------------------------- Faults -------------------------------------------------------*)

EDM_Fault:= (N03.Q.0 AND Valve1_Off) OR
			(NOT N03.Q.0 AND NOT Valve1_Off) OR
			(N03.Q.1 AND Valve2_Off) OR
			(NOT N03.Q.1 AND NOT Valve1_Off);



(*-------------------------------------- Transfer Discrete Image -----------------------------------------*)
	Discrete_Image.N01:= N01;
	Discrete_Image.N02:= N02;
	Discrete_Image.N03:= N03;
	Discrete_Image.N03_STAT:= N03_STAT;
	Discrete_Image.N04_CMD:= N04_CMD;
	Discrete_Image.N04_STAT:= N04_STAT;
	(*Option Power Distribution Nodes*)
	Discrete_Image.N999_STAT:=N999_STAT;
	Discrete_Image.N999_CMD:=N999_CMD;
	Discrete_Image.N1000_STAT:=N1000_STAT;
	Discrete_Image.N1000_CMD:=N1000_CMD;
	Discrete_Image.N1001_STAT:=N1001_STAT;
	Discrete_Image.N1001_CMD:=N1001_CMD;

(*Transfer Option Variables for Display on UI*)
	Discrete_Image.Option_EP9214_Count:= FB_In.Option_EP9214_Count;

(*Transfer Commands TO Power Distribution Node Outputs*)
	(*Device Level*)
	N04_CMD.Device.Enable_Control_Via_Fieldbus:= FALSE;
	N04_CMD.Device.Global_Reset:= FB_In.Safety_RST;
	(*Channel1 Level*)
	N04_CMD.Channel1.Output_Us:= TRUE OR FB_In.Channel1_Output_Us;;
	N04_CMD.Channel1.Output_Up:= FB_In.Enable_Motion OR FB_In.Channel1_Output_Up;
	N04_CMD.Channel1.Reset_Us:= FB_In.Safety_RST OR FB_In.Channel1_Reset_Us;
	N04_CMD.Channel1.Reset_Up:= FB_In.Safety_RST OR FB_In.Channel1_Reset_Up;
	(*Channel2Level*)
	N04_CMD.Channel2.Output_Us:= TRUE OR FB_In.Channel2_Output_Us;;
	N04_CMD.Channel2.Output_Up:= FB_In.Enable_Motion OR FB_In.Channel2_Output_Up;
	N04_CMD.Channel2.Reset_Us:= FB_In.Safety_RST OR FB_In.Channel2_Reset_Us;
	N04_CMD.Channel2.Reset_Up:= FB_In.Safety_RST OR FB_In.Channel2_Reset_Up;
	(*Channel3Level*)
	N04_CMD.Channel3.Output_Us:= TRUE OR FB_In.Channel3_Output_Us;;
	N04_CMD.Channel3.Output_Up:= FB_In.Enable_Motion OR FB_In.Channel3_Output_Up;
	N04_CMD.Channel3.Reset_Us:= FB_In.Safety_RST OR FB_In.Channel3_Reset_Us;
	N04_CMD.Channel3.Reset_Up:= FB_In.Safety_RST OR FB_In.Channel3_Reset_Up;
	(*Channel4Level*)
	N04_CMD.Channel4.Output_Us:= TRUE OR FB_In.Channel4_Output_Us;
	N04_CMD.Channel4.Output_Up:= FB_In.Enable_Motion OR FB_In.Channel4_Output_Up;
	N04_CMD.Channel4.Reset_Us:= FB_In.Safety_RST OR FB_In.Channel4_Reset_Us;
	N04_CMD.Channel4.Reset_Up:= FB_In.Safety_RST OR FB_In.Channel4_Reset_Up;
	
		(*Device Level*)
	N999_CMD.Device.Enable_Control_Via_Fieldbus:= FALSE;
	N999_CMD.Device.Global_Reset:= FB_In.Safety_RST;
	(*Channel1 Level*)
	N999_CMD.Channel1.Output_Us:= TRUE;
	N999_CMD.Channel1.Output_Up:= FB_In.Enable_Motion;
	N999_CMD.Channel1.Reset_Us:= FB_In.Safety_RST;
	N999_CMD.Channel1.Reset_Up:= FB_In.Safety_RST;
	(*Channel2Level*)
	N999_CMD.Channel2.Output_Us:= TRUE;
	N999_CMD.Channel2.Output_Up:= FB_In.Enable_Motion;
	N999_CMD.Channel2.Reset_Us:= FB_In.Safety_RST;
	N999_CMD.Channel2.Reset_Up:= FB_In.Safety_RST;
	(*Channel3Level*)
	N999_CMD.Channel3.Output_Us:= TRUE;
	N999_CMD.Channel3.Output_Up:= FB_In.Enable_Motion;
	N999_CMD.Channel3.Reset_Us:= FB_In.Safety_RST;
	N999_CMD.Channel3.Reset_Up:= FB_In.Safety_RST;
	(*Channel4Level*)
	N999_CMD.Channel4.Output_Us:= TRUE;
	N999_CMD.Channel4.Output_Up:= FB_In.Enable_Motion;
	N999_CMD.Channel4.Reset_Us:= FB_In.Safety_RST;
	N999_CMD.Channel4.Reset_Up:= FB_In.Safety_RST;
	
		(*Device Level*)
	N1000_CMD.Device.Enable_Control_Via_Fieldbus:= FALSE;
	N1000_CMD.Device.Global_Reset:= FB_In.Safety_RST;
	(*Channel1 Level*)
	N1000_CMD.Channel1.Output_Us:= TRUE;
	N1000_CMD.Channel1.Output_Up:= FB_In.Enable_Motion;
	N1000_CMD.Channel1.Reset_Us:= FB_In.Safety_RST;
	N1000_CMD.Channel1.Reset_Up:= FB_In.Safety_RST;
	(*Channel2Level*)
	N1000_CMD.Channel2.Output_Us:= TRUE;
	N1000_CMD.Channel2.Output_Up:= FB_In.Enable_Motion;
	N1000_CMD.Channel2.Reset_Us:= FB_In.Safety_RST;
	N1000_CMD.Channel2.Reset_Up:= FB_In.Safety_RST;
	(*Channel3Level*)
	N1000_CMD.Channel3.Output_Us:= TRUE;
	N1000_CMD.Channel3.Output_Up:= FB_In.Enable_Motion;
	N1000_CMD.Channel3.Reset_Us:= FB_In.Safety_RST;
	N1000_CMD.Channel3.Reset_Up:= FB_In.Safety_RST;
	(*Channel4Level*)
	N1000_CMD.Channel4.Output_Us:= TRUE;
	N1000_CMD.Channel4.Output_Up:= FB_In.Enable_Motion;
	N1000_CMD.Channel4.Reset_Us:= FB_In.Safety_RST;
	N1000_CMD.Channel4.Reset_Up:= FB_In.Safety_RST;
		
		(*Device Level*)
	N1001_CMD.Device.Enable_Control_Via_Fieldbus:= FALSE;
	N1001_CMD.Device.Global_Reset:= FB_In.Safety_RST;
	(*Channel1 Level*)
	N1001_CMD.Channel1.Output_Us:= TRUE;
	N1001_CMD.Channel1.Output_Up:= FB_In.Enable_Motion;
	N1001_CMD.Channel1.Reset_Us:= FB_In.Safety_RST;
	N1001_CMD.Channel1.Reset_Up:= FB_In.Safety_RST;
	(*Channel2Level*)
	N1001_CMD.Channel2.Output_Us:= TRUE;
	N1001_CMD.Channel2.Output_Up:= FB_In.Enable_Motion;
	N1001_CMD.Channel2.Reset_Us:= FB_In.Safety_RST;
	N1001_CMD.Channel2.Reset_Up:= FB_In.Safety_RST;
	(*Channel3Level*)
	N1001_CMD.Channel3.Output_Us:= TRUE;
	N1001_CMD.Channel3.Output_Up:= FB_In.Enable_Motion;
	N1001_CMD.Channel3.Reset_Us:= FB_In.Safety_RST;
	N1001_CMD.Channel3.Reset_Up:= FB_In.Safety_RST;
	(*Channel4Level*)
	N1001_CMD.Channel4.Output_Us:= TRUE;
	N1001_CMD.Channel4.Output_Up:= FB_In.Enable_Motion;
	N1001_CMD.Channel4.Reset_Us:= FB_In.Safety_RST;
	N1001_CMD.Channel4.Reset_Up:= FB_In.Safety_RST;

END_FUNCTION_BLOCK

// ---- POUs/FBs/FB_GTAC_ESW_20150814.TcPOU
(*FB used to Handle Enable Switch Plate I/O

------------------------------------------------------------------------
REVISION NOTES:
	Original Author(s): b.lekx-toniolo of Sodecia GTAC (broken out from Original grouped FB created by r.remillard); 
	Version 2015
		- Broke out from originally grouped "WS" FB, b.lekx-toniolo
------------------------------------------------------------------------
*)

FUNCTION_BLOCK FB_GTAC_ESW_20150814

VAR_INPUT

	Prev_EcatNode_Present: BOOL;

END_VAR

VAR

	N01 AT %I*: udt_EP1908_002;

(*Node States*)
	DiscreteNode_OK: BOOL;
	EP1908_NotPresent: BOOL;
	EP1908_PortB_MissingLink: BOOL;

(*Cable Break States*)
	ECatSlave_Cable_Breaks: UDINT;

END_VAR

VAR_OUTPUT

	EStopOK: BOOL;
	Enabling_Switch_On: BOOL;
	Disabling_Key_OK: BOOL;
	Enabling_Switch_Active: BOOL;
	Discrete_Image: udt_ESWxx_Image_20150814;



END_VAR

(*$$$$$$$$$$$$$$$$$$$$$$$$$$$$$$$$$$$$$$$$$$$$$$$$Gather Status Of Hardware $$$$$$$$$$$$$$$$$$$$$$$$$$$$$$$$$$$$$$$$$$$$$$$$$$$$*)
	(*Enable Switch Discrete I/O Nodes*)
	IF N01.InfoData.State=8
		THEN
			DiscreteNode_OK:=TRUE;
	ELSE
			DiscreteNode_OK:=FALSE;
	END_IF;


	(*Enable Switch Plate Cable Break Detection*)
	IF N01.InfoData.State=257 (*State Machine for Slave Not Present AND Previous Node is Present*)
		THEN EP1908_NotPresent:= TRUE;
	ELSE EP1908_NotPresent:= FALSE;
	END_IF;

	IF N01.InfoData.State=9224 (*Missing link, Port B*)
		THEN EP1908_PortB_MissingLink:= TRUE;
	ELSE EP1908_PortB_MissingLink:= FALSE;
	END_IF;

EcatSlave_Cable_Breaks.0:= EP1908_NotPresent AND Prev_EcatNode_Present;
EcatSlave_Cable_Breaks.1:= EP1908_PortB_MissingLink;

(*----------------------------------------------------- Map I/O---------------------------------------------*)

(*EP1908*)
EStopOK:= N01.I.0 AND N01.I.1;
Enabling_Switch_On:= N01.I.2 AND N01.I.3;
Disabling_Key_OK:= N01.I.4 AND N01.I.5;
Enabling_Switch_Active:= NOT N01.I.6 OR NOT N01.I.7;

(*Transfer Discrete Image*)
Discrete_Image.N01:= N01;

END_FUNCTION_BLOCK

// ---- POUs/FBs/FB_Emhart_20200113.TcPOU
(*
Emhart Stud Welder FB
--------------------------------------------------------------------------
REVISION NOTES
	Version 20151208:
		- Initial Concept, b.lekx-toniolo, j.underhill
		- Initial concept was only developed to get STxx safety interface up and running, further development required!!!!!
	Version 20180204
		- changed udt references to newer types. j.vandongen
	Version 20190924
		- updated instance
	Version 20200113
		- updated instance for new Profibus Mapping (TE1500 controller), j.underhill

--------------------------------------------------------------------------
*)

FUNCTION_BLOCK FB_Emhart_20200113

	VAR_INPUT
		Safety_RST					:BOOL;	(*Used to reset TwinSAFE Faults*)
		Enable_Motion				:BOOL;
		Prev_EcatNode_Present		:BOOL;

		Schedule_Select				:UINT;
		Mode_Select					:BYTE;
		Tool_Change_Mode			:BOOL;

		Restart						:BOOL;
		Weld_On					:BOOL;
		Force_WeldComp				:BOOL;
		Motion_Release_REQ			:BOOL;	(*Used with LMR Heads Only*)

		Head1_StartWeld				:BOOL;
		Head2_StartWeld				:BOOL;
		Head3_StartWeld				:BOOL;
		Head4_StartWeld				:BOOL;
		Head5_StartWeld				:BOOL;

		Head1_StartFeed				:BOOL;
		Head2_StartFeed				:BOOL;
		Head3_StartFeed				:BOOL;
		Head4_StartFeed				:BOOL;
		Head5_StartFeed				:BOOL;

		(*Used with LMR Heads Only*)
		Head1_To_WeldPos			:BOOL;
		Head2_To_WeldPos			:BOOL;
		Head3_To_WeldPos			:BOOL;
		Head4_To_WeldPos			:BOOL;
		Head5_To_WeldPos			:BOOL;

		(*Used with LMR Heads Only*)
		Head1_To_PickPos			:BOOL;
		Head2_To_PickPos			:BOOL;
		Head3_To_PickPos			:BOOL;
		Head4_To_PickPos			:BOOL;
		Head5_To_PickPos			:BOOL;

		Head1_WeldComplete_RST	:BOOL;	(*Reset Weld Complete*)
		Head2_WeldComplete_RST	:BOOL;	(*Reset Weld Complete*)
		Head3_WeldComplete_RST	:BOOL;	(*Reset Weld Complete*)
		Head4_WeldComplete_RST	:BOOL;	(*Reset Weld Complete*)
		Head5_WeldComplete_RST	:BOOL;	(*Reset Weld Complete*)

	END_VAR

	VAR
(*Hardware Data Types*)
		(*Develop Discrete Nodes*)
		T01 AT %I*					:udt_EK1100;						(*Ecat Bus Coupler*)
		T02_STAT AT %I*				:udt_EL6900_STAT_20160426;		(*EL Safety CPU status*)
		T02_CMD AT %Q*				:udt_EL6900_CMD_20121204;		(*EL Safety CPU command*)
		T03 AT %I*					:udt_EL1904_v2;					(*EL Safety Inputs*)
		T04 AT %I*					:udt_EL2904RO_v2;				(*EL Safety Outputs, Set to "I" as this terminal is safety rated, therefore read only!*)
		T05 AT %I*					:udt_EL6731;						(*EL ProfiBus Master*)

		(*Develop Profibus Node*)
		In_From_ProfiNode AT %I*		:udt_Emhart_TE1500_Input;
		Out_To_ProfiNode AT %Q*		:udt_Emhart_TE1500_Output;

		(* Nodes States*)
		DiscreteNode_OK				:BOOL;
		ProfiNode_OK				:BOOL;

		(*Cable Break Warning Flags*)
		ECatSlave_Cable_Breaks		:UDINT;
		EK1100_NotPresent 			:BOOL;			(*Coupler is Not Present on Bus when expected*)
		EK1100_PortC_MissingLink		:BOOL;  			(*Port C of EK1100 is OUT*)

		(*Safety Internals*)
		Estop_Relays_On				:BOOL;			(*Robot Estop Relays Are On, See Rxx Print Package, Page P05 and P08 *)
		Estop_Relays_Off				:BOOL;			(*Robot Estop Relays Are Off*)

		(*Standard Internals*)
		Faulted						:BOOL;

		Head1_CompleteDelay		:TON;			(*Capture Weld Complete*)
		Head2_CompleteDelay		:TON;			(*Capture Weld Complete*)
		Head3_CompleteDelay		:TON;			(*Capture Weld Complete*)
		Head4_CompleteDelay		:TON;			(*Capture Weld Complete*)
		Head5_CompleteDelay		:TON;			(*Capture Weld Complete*)


	END_VAR

	VAR_OUTPUT
		FB_Ok						:BOOL;
		(*Visualization Outputs*)
		Input_Image					:udt_Emhart_TE1500_Input;
		Output_Image					:udt_Emhart_TE1500_Output;
		Discrete_Image				:udt_STxx_DiscreteNode_20200212;

		Ready_Auto					:BOOL;
		Ready_Weld					:BOOL;
		Maint_Required				:BOOL;
		Studs_Low					:BOOL;
		Move_Clear_REQ				:BOOL;	(*Used with LMR Heads Only*)
		Motion_Release_ACK			:BOOL;	(*Used with LMR Heads Only*)

		Fault_Grp_Bit0				:BOOL;
		Fault_Grp_Bit1				:BOOL;
		Fault_Grp_Bit2				:BOOL;

		Fault_Code_Bit0				:BOOL;
		Fault_Code_Bit1				:BOOL;
		Fault_Code_Bit2				:BOOL;
		Fault_Code_Bit3				:BOOL;
		Fault_Code_Bit4				:BOOL;
		Fault_Code_Bit5				:BOOL;
		Fault_Code_Bit6				:BOOL;
		Fault_Code_Bit7				:BOOL;
		Fault_Code_Bit8				:BOOL;

		Head1_Faulted				:BOOL;
		Head1_WeldComp			:BOOL;
		Head1_Back					:BOOL;
		Head1_SOW					:BOOL;	(*SOW = Stud On Workpiece*)
		Head1_In_Tolerance			:BOOL;
		Head1_LMR_Connected		:BOOL;	(*Used with LMR Heads Only*)
		Head1_In_WeldPos			:BOOL;	(*Used with LMR Heads Only*)
		Head1_In_PickPos			:BOOL;	(*Used with LMR Heads Only*)
		Head1_Stud_Gripper			:BOOL;	(*Used with LMR Heads Only*)
		Head1_Weld_Completed		:BOOL;

		Head2_Faulted				:BOOL;
		Head2_WeldComp			:BOOL;
		Head2_Back					:BOOL;
		Head2_SOW					:BOOL;	(*SOW = Stud On Workpiece*)
		Head2_In_Tolerance			:BOOL;
		Head2_LMR_Connected		:BOOL;	(*Used with LMR Heads Only*)
		Head2_In_WeldPos			:BOOL;	(*Used with LMR Heads Only*)
		Head2_In_PickPos			:BOOL;	(*Used with LMR Heads Only*)
		Head2_Stud_Gripper			:BOOL;	(*Used with LMR Heads Only*)
		Head2_Weld_Completed		:BOOL;

		Head3_Faulted				:BOOL;
		Head3_WeldComp			:BOOL;
		Head3_Back					:BOOL;
		Head3_SOW					:BOOL;	(*SOW = Stud On Workpiece*)
		Head3_In_Tolerance			:BOOL;
		Head3_LMR_Connected		:BOOL;	(*Used with LMR Heads Only*)
		Head3_In_WeldPos			:BOOL;	(*Used with LMR Heads Only*)
		Head3_In_PickPos			:BOOL;	(*Used with LMR Heads Only*)
		Head3_Stud_Gripper			:BOOL;	(*Used with LMR Heads Only*)
		Head3_Weld_Completed		:BOOL;

		Head4_Faulted				:BOOL;
		Head4_WeldComp			:BOOL;
		Head4_Back					:BOOL;
		Head4_SOW					:BOOL;	(*SOW = Stud On Workpiece*)
		Head4_In_Tolerance			:BOOL;
		Head4_LMR_Connected		:BOOL;	(*Used with LMR Heads Only*)
		Head4_In_WeldPos			:BOOL;	(*Used with LMR Heads Only*)
		Head4_In_PickPos			:BOOL;	(*Used with LMR Heads Only*)
		Head4_Stud_Gripper			:BOOL;	(*Used with LMR Heads Only*)
		Head4_Weld_Completed		:BOOL;

		Head5_Faulted				:BOOL;
		Head5_WeldComp			:BOOL;
		Head5_Back					:BOOL;
		Head5_SOW					:BOOL;	(*SOW = Stud On Workpiece*)
		Head5_In_Tolerance			:BOOL;
		Head5_LMR_Connected		:BOOL;	(*Used with LMR Heads Only*)
		Head5_In_WeldPos			:BOOL;	(*Used with LMR Heads Only*)
		Head5_In_PickPos			:BOOL;	(*Used with LMR Heads Only*)
		Head5_Stud_Gripper			:BOOL;	(*Used with LMR Heads Only*)
		Head5_Weld_Completed		:BOOL;

	END_VAR

	(*Set FB_OK to True*)
	FB_OK:= TRUE;
(*$$$$$$$$$$$$$$$$$$$$$$$$$$$$$$$$$$$$$$$$$$$$$$$$Gather Status Of Hardware $$$$$$$$$$$$$$$$$$$$$$$$$$$$$$$$$$$$$$$$$$$$$$$$$$$$*)
	(*Discrete I/O Node*)
	IF (T01.InfoData.State=8) AND (T02_Stat.InfoData.State=8) AND (T03.InfoData.State=8) AND (T04.InfoData.State=8) AND (T05.InfoData.State=8)
		THEN DiscreteNode_OK:=TRUE;
	ELSE DiscreteNode_OK:=FALSE;
	END_IF


	(*Develop Port Connection Warning Flags*)
	IF T01.InfoData.State=257 (*State Machine for Slave Not Present*)
		THEN EK1100_NotPresent:= TRUE;
	ELSE EK1100_NotPresent := FALSE;
	END_IF

	IF T01.InfoData.State=17416 (*State Machine for Link Missing at Port C*)
		THEN EK1100_PortC_MissingLink:= TRUE; (*PortC is OUT Port*)
	ELSE EK1100_PortC_MissingLink := FALSE;
	END_IF


	(*Profibus Node*)
	IF In_From_ProfiNode.Inputs.DpState=0
		THEN ProfiNode_OK:=TRUE;
	ELSE ProfiNode_OK:=FALSE;
	END_IF;

	(*Wrap up break Flags to Variable for shipment to UI*)
	ECatSlave_Cable_Breaks.0:= EK1100_NotPresent AND Prev_EcatNode_Present;
	ECatSlave_Cable_Breaks.1:= EK1100_PortC_MissingLink;
	ECatSlave_Cable_Breaks.16:= (In_From_Profinode.Inputs.DpState=2);		(*Cable Break Possible from EL6731 to Profibus Slave Care in Nelson Stud Controller*)

(*$$$$$$$$$$$$$$$$$$$$$$$$$$$$$$$$$$$$$$$$$$$$$ Gather Safety Inputs $$$$$$$$$$$$$$$$$$$$$$$$$$$$$$$$$$$$$$$$$$$$$$$$$$$$$$$$$*)

	Estop_Relays_On:= NOT T03.I.0 AND T04.Q.0 AND T04.Q.1;
	Estop_Relays_Off:= T03.I.0;

(*$$$$$$$$$$$$$$$$$$$$$$$$$$$$$$$$$$$$$$$$$$$$$ Gather Standard Inputs  (From Stud Controller Outputs $$$$$$$$$$$$$$$$$$$$$$$$$$$$$$$$$$$$$$$$$$$$$$$$$$$$$$$$$*)

	(*-------- Profibus Inputs from Controller -----------*)

	Head1_Faulted:= 			NOT In_From_ProfiNode.Byte0.0;	(*Signal from TE1500 is "No Fault"*)
	Head1_WeldComp:=		In_From_ProfiNode.Byte0.1;
	Head1_Back:= 			In_From_ProfiNode.Byte0.2;
	Head1_SOW:=			In_From_ProfiNode.Byte0.3;
	Head1_In_Tolerance:=		In_From_ProfiNode.Byte0.4;

	Head2_Faulted:= 			NOT In_From_ProfiNode.Byte0.5;	(*Signal from TE1500 is "No Fault"*)
	Head2_WeldComp:=		In_From_ProfiNode.Byte0.6;
	Head2_Back:= 			In_From_ProfiNode.Byte0.7;
	Head2_SOW:=			In_From_ProfiNode.Byte1.0;
	Head2_In_Tolerance:=		In_From_ProfiNode.Byte1.1;

	Head3_Faulted:= 			NOT In_From_ProfiNode.Byte1.2;	(*Signal from TE1500 is "No Fault"*)
	Head3_WeldComp:=		In_From_ProfiNode.Byte1.3;
	Head3_Back:= 			In_From_ProfiNode.Byte1.4;
	Head3_SOW:=			In_From_ProfiNode.Byte1.5;
	Head3_In_Tolerance:=		In_From_ProfiNode.Byte1.6;

	Head4_Faulted:= 			NOT In_From_ProfiNode.Byte1.7;	(*Signal from TE1500 is "No Fault"*)
	Head4_WeldComp:=		In_From_ProfiNode.Byte2.0;
	Head4_Back:= 			In_From_ProfiNode.Byte2.1;
	Head4_SOW:=			In_From_ProfiNode.Byte2.2;
	Head4_In_Tolerance:=		In_From_ProfiNode.Byte2.3;

	Head5_Faulted:= 			NOT In_From_ProfiNode.Byte2.4;	(*Signal from TE1500 is "No Fault"*)
	Head5_WeldComp:=		In_From_ProfiNode.Byte2.5;
	Head5_Back:= 			In_From_ProfiNode.Byte2.6;
	Head5_SOW:=			In_From_ProfiNode.Byte2.7;
	Head5_In_Tolerance:=		In_From_ProfiNode.Byte3.0;

	Maint_Required:=			In_From_ProfiNode.Byte3.1;
	Studs_Low:=				In_From_ProfiNode.Byte3.2;
	Ready_Auto:=			In_From_ProfiNode.Byte3.3;
	Ready_Weld:=			In_From_ProfiNode.Byte3.4;

	Fault_Grp_Bit0:=			In_From_ProfiNode.Byte3.5;
	Fault_Grp_Bit1:=			In_From_ProfiNode.Byte3.6;
	Fault_Grp_Bit2:=			In_From_ProfiNode.Byte3.7;

	Fault_Code_Bit0:=			In_From_ProfiNode.Byte4.0;
	Fault_Code_Bit1:=			In_From_ProfiNode.Byte4.1;
	Fault_Code_Bit2:=			In_From_ProfiNode.Byte4.2;
	Fault_Code_Bit3:=			In_From_ProfiNode.Byte4.3;
	Fault_Code_Bit4:=			In_From_ProfiNode.Byte4.4;
	Fault_Code_Bit5:=			In_From_ProfiNode.Byte4.5;
	Fault_Code_Bit6:=			In_From_ProfiNode.Byte4.6;
	Fault_Code_Bit7:=			In_From_ProfiNode.Byte4.7;
	Fault_Code_Bit8:=			In_From_ProfiNode.Byte5.0;
											(*Byte5.1 - Reserved*)

	(*NOTE - Below Inputs used with LMR Heads Only*)
	Move_Clear_REQ:=		In_From_ProfiNode.Byte5.2;

	Head1_LMR_Connected:=	In_From_ProfiNode.Byte5.3;
	Head2_LMR_Connected:=	In_From_ProfiNode.Byte5.4;
	Head3_LMR_Connected:=  	In_From_ProfiNode.Byte5.5;
	Head4_LMR_Connected:=  	In_From_ProfiNode.Byte5.6;
	Head5_LMR_Connected:=	In_From_ProfiNode.Byte5.7;

	Head1_In_WeldPos:=		In_From_ProfiNode.Byte6.0;
	Head2_In_WeldPos:=		In_From_ProfiNode.Byte6.1;
	Head3_In_WeldPos:=		In_From_ProfiNode.Byte6.2;
	Head4_In_WeldPos:=		In_From_ProfiNode.Byte6.3;
	Head5_In_WeldPos:=		In_From_ProfiNode.Byte6.4;

	Head1_In_PickPos:=		In_From_ProfiNode.Byte6.5;
	Head2_In_PickPos:=		In_From_ProfiNode.Byte6.6;
	Head3_In_PickPos:=		In_From_ProfiNode.Byte6.7;
	Head4_In_PickPos:=		In_From_ProfiNode.Byte7.0;
	Head5_In_PickPos:=		In_From_ProfiNode.Byte7.1;

	Head1_Stud_Gripper:= 	In_From_ProfiNode.Byte7.2;
	Head2_Stud_Gripper:= 	In_From_ProfiNode.Byte7.3;
	Head3_Stud_Gripper:= 	In_From_ProfiNode.Byte7.4;
	Head4_Stud_Gripper:= 	In_From_ProfiNode.Byte7.5;
	Head5_Stud_Gripper:= 	In_From_ProfiNode.Byte7.6;

	Motion_Release_ACK:=	In_From_ProfiNode.Byte7.7;




(*$$$$$$$$$$$$$$$$$$$$$$$$$$$$$$$$$$$$$$$$$$$$$$$$ Internal Code $$$$$$$$$$$$$$$$$$$$$$$$$$$$$$$$$$$$$$$$$$$$$$$$$$$$$$$$$$$$$$$$$$$$*)

	(*Capture Weld Complete - Head 1*)
	Head1_CompleteDelay.PT:= T#500ms;
	Head1_CompleteDelay.IN:= Head1_WeldComp AND Head1_Back AND Head1_In_Tolerance;
	Head1_CompleteDelay();

	IF Head1_CompleteDelay.Q
		THEN Head1_Weld_Completed:= TRUE;
	ELSIF Head1_WeldComplete_RST
		THEN Head1_Weld_Completed:= FALSE;
	END_IF;

	(*Capture Weld Complete - Head 2*)
	Head2_CompleteDelay.PT:= T#500ms;
	Head2_CompleteDelay.IN:= Head2_WeldComp AND Head2_Back AND Head2_In_Tolerance;
	Head2_CompleteDelay();

	IF Head2_CompleteDelay.Q
		THEN Head2_Weld_Completed:= TRUE;
	ELSIF Head2_WeldComplete_RST
		THEN Head2_Weld_Completed:= FALSE;
	END_IF;

	(*Capture Weld Complete - Head 3*)
	Head3_CompleteDelay.PT:= T#500ms;
	Head3_CompleteDelay.IN:= Head3_WeldComp AND Head3_Back AND Head3_In_Tolerance;
	Head3_CompleteDelay();

	IF Head3_CompleteDelay.Q
		THEN Head3_Weld_Completed:= TRUE;
	ELSIF Head3_WeldComplete_RST
		THEN Head3_Weld_Completed:= FALSE;
	END_IF;

	(*Capture Weld Complete - Head 4*)
	Head4_CompleteDelay.PT:= T#500ms;
	Head4_CompleteDelay.IN:= Head4_WeldComp AND Head4_Back AND Head4_In_Tolerance;
	Head4_CompleteDelay();

	IF Head4_CompleteDelay.Q
		THEN Head4_Weld_Completed:= TRUE;
	ELSIF Head4_WeldComplete_RST
		THEN Head4_Weld_Completed:= FALSE;
	END_IF;

	(*Capture Weld Complete - Head 5*)
	Head5_CompleteDelay.PT:= T#500ms;
	Head5_CompleteDelay.IN:= Head5_WeldComp AND Head5_Back AND Head5_In_Tolerance;
	Head5_CompleteDelay();

	IF Head5_CompleteDelay.Q
		THEN Head5_Weld_Completed:= TRUE;
	ELSIF Head5_WeldComplete_RST
		THEN Head5_Weld_Completed:= FALSE;
	END_IF;



(*$$$$$$$$$$$$$$$$$$$$$$$$$$$$$$$$$$$$$$$$$$$$$$$$$$$ Faults $$$$$$$$$$$$$$$$$$$$$$$$$$$$$$$$$$$$$$$$$$$$$$$$$$$$$$$*)

	Faulted := (Head1_Faulted OR
				Head2_Faulted OR
				Head3_Faulted OR
				Head4_Faulted OR
				Head5_Faulted OR
				NOT Ready_Auto);


(*$$$$$$$$$$$$$$$$$$$$$$$$$$$$$$$$$$$$$$$$$$$$$$ Transfer Standard Outputs $$$$$$$$$$$$$$$$$$$$$$$$$$$$$$$$$$$$$$$$$$$*)

	(*Transfer Profibus I/O Image*)
	Input_Image.Inputs.DpState:= In_From_ProfiNode.Inputs.DpState;
	Input_Image.Inputs.ExtDiagFlag:= In_From_ProfiNode.Inputs.ExtDiagFlag;

	Input_Image.Byte0:= In_From_ProfiNode.Byte0;
	Input_Image.Byte1:= In_From_ProfiNode.Byte1;
	Input_Image.Byte2:= In_From_ProfiNode.Byte2;
	Input_Image.Byte3:= In_From_ProfiNode.Byte3;
	Input_Image.Byte4:= In_From_ProfiNode.Byte4;
	Input_Image.Byte5:= In_From_ProfiNode.Byte5;
	Input_Image.Byte6:= In_From_ProfiNode.Byte6;
	Input_Image.Byte7:= In_From_ProfiNode.Byte7;

	Output_Image.Byte0:= Out_To_ProfiNode.Byte0;
	Output_Image.Byte1:= Out_To_ProfiNode.Byte1;
	Output_Image.Byte2:= Out_To_ProfiNode.Byte2;
	Output_Image.Byte3:= Out_To_ProfiNode.Byte3;
	Output_Image.Byte4:= Out_To_ProfiNode.Byte4;
	Output_Image.Byte5:= Out_To_ProfiNode.Byte5;
	Output_Image.Byte6:= Out_To_ProfiNode.Byte6;
	Output_Image.Byte7:= Out_To_ProfiNode.Byte7;

	(*Transfer Discrete I/O Image*)
	Discrete_Image.T01:=T01;
	Discrete_Image.T02_STAT:=T02_STAT;
	Discrete_Image.T03:=T03;
	Discrete_Image.T04:=T04;
	Discrete_Image.T05:=T05;
	Discrete_Image.Profinode_Stat:=In_From_ProfiNode.Inputs;

	(*-------- Profibus Outputs to Controller -----------*)

	(*Out To Emhart Input Byte0*)
	Out_To_ProfiNode.Byte0.0:= Enable_Motion AND Head1_StartWeld;		(*Head 1 Start Weld*)
	Out_To_ProfiNode.Byte0.1:= Enable_Motion AND Head2_StartWeld;		(*Head 2 Start Weld*)
	Out_To_ProfiNode.Byte0.2:= Enable_Motion AND Head3_StartWeld;		(*Head 3 Start Weld*)
	Out_To_ProfiNode.Byte0.3:= Enable_Motion AND Head4_StartWeld;		(*Head 4 Start Weld*)
	Out_To_ProfiNode.Byte0.4:= Enable_Motion AND Head5_StartWeld;		(*Head 5 Start Weld*)
	Out_To_ProfiNode.Byte0.5:= Enable_Motion AND Head1_StartFeed;		(*Head 1 Start Feed*)
	Out_To_ProfiNode.Byte0.6:= Enable_Motion AND Head2_StartFeed;		(*Head 2 Start Feed*)
	Out_To_ProfiNode.Byte0.7:= Enable_Motion AND Head3_StartFeed;		(*Head 3 Start Feed*)

	(*Out To Emhart Input Byte1*)
	Out_To_ProfiNode.Byte1.0:= Enable_Motion AND Head4_StartFeed;		(*Head 4 Start Feed*)
	Out_To_ProfiNode.Byte1.1:= Enable_Motion AND Head5_StartFeed;		(*Head 5 Start Feed*)
	Out_To_ProfiNode.Byte1.2:= Schedule_Select.0;						(*Schedule Select Bit0*)
	Out_To_ProfiNode.Byte1.3:= Schedule_Select.1;						(*Schedule Select Bit1*)
	Out_To_ProfiNode.Byte1.4:= Schedule_Select.2;						(*Schedule Select Bit2*)
	Out_To_ProfiNode.Byte1.5:= Schedule_Select.3;						(*Schedule Select Bit3*)
	Out_To_ProfiNode.Byte1.6:= Schedule_Select.4;						(*Schedule Select Bit4*)
	Out_To_ProfiNode.Byte1.7:= Schedule_Select.5;						(*Schedule Select Bit5*)

	(*Out To Emhart Input Byte2*)
	Out_To_ProfiNode.Byte2.0:= Schedule_Select.6;						(*Schedule Select Bit6*)
	Out_To_ProfiNode.Byte2.1:= FALSE;									(*Reserved*)
	Out_To_ProfiNode.Byte2.2:= Enable_Motion AND Restart;				(*Restart Weld*)
	Out_To_ProfiNode.Byte2.3:= Force_WeldComp;						(*Force Weld Complete*)
	Out_To_ProfiNode.Byte2.4:= Mode_Select.0;							(*Mode Select Bit0*)
	Out_To_ProfiNode.Byte2.5:= Mode_Select.1;							(*Mode Select Bit1*)
	Out_To_ProfiNode.Byte2.6:= Tool_Change_Mode;						(*Tool Change Mode*)
	Out_To_ProfiNode.Byte2.7:= FALSE;									(*Reserved*)

	(*Out To Emhart Input Byte3 - ALL RESERVED*)
	Out_To_ProfiNode.Byte3.0:= FALSE;
	Out_To_ProfiNode.Byte3.1:= FALSE;
	Out_To_ProfiNode.Byte3.2:= FALSE;
	Out_To_ProfiNode.Byte3.3:= FALSE;
	Out_To_ProfiNode.Byte3.4:= FALSE;
	Out_To_ProfiNode.Byte3.5:= FALSE;
	Out_To_ProfiNode.Byte3.6:= FALSE;
	Out_To_ProfiNode.Byte3.7:= FALSE;

	(*Out To Emhart Input Byte4 - ALL RESERVED*)
	Out_To_ProfiNode.Byte4.0:= FALSE;
	Out_To_ProfiNode.Byte4.1:= FALSE;
	Out_To_ProfiNode.Byte4.2:= FALSE;
	Out_To_ProfiNode.Byte4.3:= FALSE;
	Out_To_ProfiNode.Byte4.4:= FALSE;
	Out_To_ProfiNode.Byte4.5:= FALSE;
	Out_To_ProfiNode.Byte4.6:= FALSE;
	Out_To_ProfiNode.Byte4.7:= FALSE;

	(*Out To Emhart Input Byte5 - ALL RESERVED*)
	Out_To_ProfiNode.Byte5.0:= FALSE;
	Out_To_ProfiNode.Byte5.1:= FALSE;
	Out_To_ProfiNode.Byte5.2:= FALSE;
	Out_To_ProfiNode.Byte5.3:= FALSE;
	Out_To_ProfiNode.Byte5.4:= FALSE;
	Out_To_ProfiNode.Byte5.5:= FALSE;
	Out_To_ProfiNode.Byte5.6:= FALSE;
	Out_To_ProfiNode.Byte5.7:= FALSE;

	(*Out To Emhart Input Byte6*)
	Out_To_ProfiNode.Byte6.0:= Enable_Motion AND Head1_To_WeldPos;		(*Head 1 To Weld Position*)
	Out_To_ProfiNode.Byte6.1:= Enable_Motion AND Head2_To_WeldPos;		(*Head 2 To Weld Position*)
	Out_To_ProfiNode.Byte6.2:= Enable_Motion AND Head3_To_WeldPos;		(*Head 3 To Weld Position*)
	Out_To_ProfiNode.Byte6.3:= Enable_Motion AND Head4_To_WeldPos;		(*Head 4 To Weld Position*)
	Out_To_ProfiNode.Byte6.4:= Enable_Motion AND Head5_To_WeldPos;		(*Head 5 To Weld Position*)
	Out_To_ProfiNode.Byte6.5:= Enable_Motion AND Head1_To_PickPos;		(*Head 1 To Pickup Position*)
	Out_To_ProfiNode.Byte6.6:= Enable_Motion AND Head2_To_PickPos;		(*Head 2 To Pickup Position*)
	Out_To_ProfiNode.Byte6.7:= Enable_Motion AND Head3_To_PickPos;		(*Head 3 To Pickup Position*)

	(*Out To Emhart Input Byte7*)
	Out_To_ProfiNode.Byte7.0:= Enable_Motion AND Head4_To_PickPos;		(*Head 4 To Pickup Position*)
	Out_To_ProfiNode.Byte7.1:= Enable_Motion AND Head5_To_PickPos;		(*Head 5 To Pickup Position*)
	Out_To_ProfiNode.Byte7.2:= FALSE;										(*Reserved*)
	Out_To_ProfiNode.Byte7.3:= FALSE;										(*Reserved*)
	Out_To_ProfiNode.Byte7.4:= FALSE;										(*Reserved*)
	Out_To_ProfiNode.Byte7.5:= FALSE;										(*Reserved*)
	Out_To_ProfiNode.Byte7.6:= FALSE;										(*Reserved*)
	Out_To_ProfiNode.Byte7.7:= Motion_Release_REQ;						(*Motion Release*)

(*$$$$$$$$$$$$$$$$$$$$$$$$$$$$$$$$$$$$$$$$$$$$$$ Transfer Safety Outputs $$$$$$$$$$$$$$$$$$$$$$$$$$$$$$$$$$$$$$$$$$$*)
	(*Set All Safety Groups to Run*)
		T02_CMD.SGs_RUNSTOP:= TRUE;
	(*Reset Of Safety Group Errors*)
		T02_CMD.SGs_ERRAck:= Safety_RST;
	(*Reset Only Used FBs With In Safety Group*)
		(*Reset of Estop, Safety Gate and Misc FBs*)
		T02_CMD.FBs_ControlPowerPB:= Safety_RST;

END_FUNCTION_BLOCK

// ---- POUs/FBs/FB_Graco_Seal_20200716.TcPOU
(*Function block created for Graco Sealer*)
(*July 31 2014*)
(*Rev1 - JVD initial creation*)
(*
------------------------------------------------------------------------------------------
	REVISION NOTES:
	Version 20141017:
	- Added Error_Reset and Dry_Cycle FB Inputs to remove dependancies on external variable, b.lekx-toniolo
	Version 20141127:
	- Added ability to map Internal or External EL6731 Proibus Master, b.lekx-toniolo
	Version 20141209
	- General Structure Clean-up, b.lekx-toniolo
	Version 20160302
	- Added purge function, JVD
	- Added Enable_Motion, JVD
	-Added All_SafetiesOK, JVD
	-Added Faulted to the reset bit, JVD
	Version 20160405
	- added Disp1_No_Error to Faulted, JVD
	-added ProfiNode_OK to Fault, JVD
	Version 20160412
	- re-mapped purge to style select 15 at request of Graco for better table updates, blt
	Version 20161202
	-develop code for up to 4 dispense heads, j.vandongen
	-added capture for sealant/volume Ok, j.vandongen
	Version 20170227
	-fixed copy/paste typos, jvandongen
	Version 20171201
	- fixed option gun count comparissons in the code, j.vandongen
	Version 20200716
	- changed from PCF to iQ controls (new GSD map), j.vandongen

------------------------------------------------------------------------------------------
*)
FUNCTION_BLOCK FB_Graco_Seal_20200716

	VAR_INPUT
		External_Terminal_Enable: BOOL; (* Set Bit Low if you will be using the Internal Profibus Master Terminal Instance, set High to Pass Profibus Master Data from External*)
		Txx_External_ProfiMaster: udt_EL6731;

		Enable_Motion: BOOL;
		All_SafetiesOK: BOOL;
		Dry_Cycle: BOOL;

		(*Inputs into FB for Option Selection*)
		Option_Tandem: BOOL;
		Option_Heat1: BOOL;
		Option_Heat2: BOOL;


		(*Inputs to FB to Control Sealer System*)
		Error_Reset: BOOL;




		(*Pump 1- Inputs from Graco*)
		Pump1_HeartBeat: BOOL;
		Pump1_Control_Ready: BOOL;
		Pump1_System_Active: BOOL;
		Pump1_Control_Active: BOOL;
		Pump1_NoAlarms_Active: BOOL;
		Pump1_NoDeviations_Active: BOOL;
		Pump1_NoAdvisory_Active: BOOL;
		Pump1_Ready_To_Dispense: BOOL;

		Pump1_PreCharge_Active: BOOL;
		Pump1_Dispense_In_Process: BOOL;
		Pump1_Drum_Low: BOOL;
		Pump1_Drum_Empty: BOOL;
		Pump1_Not_Primed: BOOL;
		Pump1_In_Job_Cycle: BOOL;
		Pump1_Prime_Active: BOOL;
		Pump1_Valve_Depressurization_Active: BOOL;

		Pump1_Platen_Depressurization_Active: BOOL;
		Pump1_Auto_Depressurization_Active: BOOL;
		Pump1_Auto_Depressurization_Happened: BOOL;
		Pump1_Trying_To_Move: BOOL;
		Pump1_Moving: BOOL;
		Pump1_DispenseValve_Opened: BOOL;
		Pump1_PlatenValve_Opened: BOOL;
		Pump1_Tandem_Active_Pump: BOOL; 			(*0 =Pump 1, 1 = Pump 2*)

		Pump1_EFlo_iQ_Mode_Active: BOOL;
		Pump1_ChangeOver_Occured: BOOL;
		(*Reserved Bit 1*)
		(*Reserved Bit 2*)
		(*Reserved Bit 3*)
		(*Reserved Bit 4*)
		(*Reserved Bit 5*)
		(*Reserved Bit 6*)

		Pump1_ActualPump_Flowrate: UINT;				(*xxxx cc/min*)
		Pump1_Outlet_Pressure: UINT; 					(*xxx.x bar*)
		Pump1_Valve_Pressure: UINT; 					(*xxx.x bar*)
		Pump1_Active_Style_Loaded: UINT;
		Pump1_Active_Style_Precharge: UINT; 			(*xxx.x bar*)
		Pump1_Active_Style_Flowrate: UINT; 			(*xxxx cc/min*)
		Pump1_Active_Style_ShotSize: UINT; 			(*xxx.xx cc*)
		Pump1_Actual_Amount_Dispense:UDINT; 		(*xxxx.xx cc*)
		Pump1_Actual_Shot_Size: UDINT;				(*xx.xx cc*)
		Pump1_Actual_Style_PreCharge_REQ: UINT;		(*xxx.x bar*)
		Pump1_Actual_Style_Flowrate_REQ: UINT;		(*xxxx cc/min*)
		Pump1_Actual_Style_Shot_Size_REQ: UINT;		(*xxx.xx cc*)
		Pump1_PumpPosition: UINT;					(*x.xxxx inches*)
		Pump1_Data_Exchange_Active_CMD: UINT;
		Pump1_Data_Exchange_Active_CMD_Value: UDINT;


		(*Pump 2 - Inputs Only used for Tandem systems*)
		Pump2_HeartBeat: BOOL;
		Pump2_Control_Ready: BOOL;
		Pump2_System_Active: BOOL;
		Pump2_Control_Active: BOOL;
		Pump2_NoAlarms_Active: BOOL;
		Pump2_NoDeviations_Active: BOOL;
		Pump2_NoAdvisory_Active: BOOL;
		Pump2_Ready_To_Dispense: BOOL;

		Pump2_PreCharge_Active: BOOL;
		Pump2_Dispense_In_Process: BOOL;
		Pump2_Drum_Low: BOOL;
		Pump2_Drum_Empty: BOOL;
		Pump2_Not_Primed: BOOL;
		Pump2_In_Job_Cycle: BOOL;
		Pump2_Prime_Active: BOOL;
		Pump2_Valve_Depressurization_Active: BOOL;

		Pump2_Platen_Depressurization_Active: BOOL;
		Pump2_Auto_Depressurization_Active: BOOL;
		Pump2_Auto_Depressurization_Happened: BOOL;
		Pump2_Trying_To_Move: BOOL;
		Pump2_Moving: BOOL;
		Pump2_DispenseValve_Opened: BOOL;
		Pump2_PlatenValve_Opened: BOOL;
		Pump2_Tandem_Active_Pump: BOOL; 			(*0 =Pump 1, 1 = Pump 2*)

		Pump2_EFlo_iQ_Mode_Active: BOOL;
		(*Reserved Bit 1*)
		(*Reserved Bit 2*)
		(*Reserved Bit 3*)
		(*Reserved Bit 4*)
		(*Reserved Bit 5*)
		(*Reserved Bit 6*)
		(*Reserved Bit 7*)

		Pump2_ActualPump_Flowrate: UINT;				(*xxxx cc/min*)
		Pump2_Outlet_Pressure: UINT; 					(*xxx.x bar*)
		Pump2_Data_Exchange_Active_CMD: UINT;
		Pump2_Data_Exchange_Active_CMD_Value: UDINT;


		(*Heat 1 - Inputs from Graco*)
		Heat1_Heartbeat: BOOL;
		Heat1_Enabled: BOOL;
		Heat1_Control_Active: BOOL;
		Heat1_ON: BOOL;
		Heat1_WarmingUp: BOOL;
		Heat1_At_Temp: BOOL;
		Heat1_Temp_Soak_Mode: BOOL;
		Heat1_SetBack_Mode: BOOL;

		Heat1_Off: BOOL;
		Heat1_Module_NoAlarms_Active: BOOL;
		Heat1_Module_NoDeviations_Active: BOOL;
		Heat1_Module_NoAdvisory_Active: BOOL;
		Heat1_Zone_NoAlarms_Active: BOOL;
		Heat1_Zone_NoDeviations_Active: BOOL;
		Heat1_Zone_NoAdvisory_Active: BOOL;
		Heat1_Idle_Timeout_Happened: BOOL;

		Heat1_Soak_Time_Remaining: UINT;	(*xx seconds*)
		Heat1_Data_Exchange_Active_CMD: UINT;
		Heat1_Data_Exchange_Active_CMD_Value: UDINT;


		(*Heat 2 - Inputs from Graco. Only used if tandem pump is on*)
		Heat2_Heartbeat: BOOL;
		Heat2_Enabled: BOOL;
		Heat2_Control_Active: BOOL;
		Heat2_ON: BOOL;
		Heat2_WarmingUp: BOOL;
		Heat2_At_Temp: BOOL;
		Heat2_Temp_Soak_Mode: BOOL;
		Heat2_SetBack_Mode: BOOL;

		Heat2_Off: BOOL;
		Heat2_Module_NoAlarms_Active: BOOL;
		Heat2_Module_NoDeviations_Active: BOOL;
		Heat2_Module_NoAdvisory_Active: BOOL;
		Heat2_Zone_NoAlarms_Active: BOOL;
		Heat2_Zone_NoDeviations_Active: BOOL;
		Heat2_Zone_NoAdvisory_Active: BOOL;
		Heat2_Idle_Timeout_Happened: BOOL;

		Heat2_Soak_Time_Remaining: UINT;	(*xx seconds*)
		Heat2_Data_Exchange_Active_CMD: UINT;
		Heat2_Data_Exchange_Active_CMD_Value: UDINT;



	END_VAR


	VAR
		Txx_Internal_ProfiMaster AT %I*: udt_EL6731;

		(*Develop Profibus Slave Node to map Profibus Slave I/O*)
		GracoSealer_Inputs AT %I*: udt_Graco_Input;
		GracoSealer_Outputs AT %Q*: udt_Graco_Outputs;

		Purge_Trigger1: TON;
		Purge_CompleteTrigger1: TON;

		DiscreteNode_OK: BOOL;
		Profinode_OK: BOOL;

		Faulted: BOOL;

		(*Status Information regarding Graco System*)




	END_VAR

	VAR_OUTPUT
		(*Output Data to External*)
		FB_OK: BOOL;

		Dispense_Amount: UINT;
		Disp1_Bypass: BOOL;
		Disp1_Faulted: BOOL;
		Disp1_Ready: BOOL;
		Disp1_Volume_NotOK: BOOL;
		Disp1_Bypass_Ack: BOOL;


		(*Pump - Ouputs*)
		Pump1_Sys_Data_Exchange_CMD: UINT;

		Pump1_Sys_Enable: BOOL;
		Pump1_Sys_Disable_REQ: BOOL;
		Pump1_Lockout: BOOL;
		Pump1_Style_Enable: BOOL;
		Pump1_Go: BOOL;
		Pump1_Disp_Complete: BOOL;
		Pump1_Tandem_Cross_REQ: BOOL;
		Pump2_Prime_Inactive_Pump_REQ: BOOL;

		Pump1_Valve_Depressurization_REQ: BOOL;
		Pump1_Platen_Depressurization_REQ: BOOL;
		Pump1_Auto_Depressurization_Cancel_REQ: BOOL;
		Pump_Acknowledge_Clear_Errors: BOOL; (*both pumps*)
		(*Reserved Bit 1*)
		(*Reserved Bit 2*)
		(*Reserved Bit 3*)
		(*Reserved Bit 4*)

		Pump1_Desired_Style_Numb: UINT;
		Pump1_Style_PreCharge_REQ: UINT;	(*xxx.x bars*)
		Pump1_FlowRate_REQ: UINT;			(*xxxx cc/min*)
		Pump1_ShotSize_REQ: UINT;			(*xxx.xx cc*)
		Pump2_PrimePressure_Target: UINT;	(*xxx.x bars*)
		Pump2_PrimeFlow_Target: UINT;			(*xxxx cc/min*)

		Heat1_HeatEnabled_REQ: BOOL;
		Heat1_HeatDissabled_REQ: BOOL;
		Heat1_PLC_Lockout: BOOL;
		Heat1_Heat_ON_REQ: BOOL;
		Heat1_Heat_OFF_REQ: BOOL;
		Heat1_Setback_REQ: BOOL;
		Heat1_Acknowledge_Clear_Errors: BOOL;
		(*Reserved Bit 1*)

		(*Reserved Bit 2*)
		(*Reserved Bit 3*)
		(*Reserved Bit 4*)
		(*Reserved Bit 5*)
		(*Reserved Bit 6*)
		(*Reserved Bit 7*)
		(*Reserved Bit 8*)

		Heat1_Data_Exchange_CMD: UINT;
		Heat1_Data_Exchange_CMD_Value: UDINT;

		Heat2_HeatEnabled_REQ: BOOL;
		Heat2_HeatDissabled_REQ: BOOL;
		Heat2_PLC_Lockout: BOOL;
		Heat2_Heat_ON_REQ: BOOL;
		Heat2_Heat_OFF_REQ: BOOL;
		Heat2_Setback_REQ: BOOL;
		Heat2_Acknowledge_Clear_Errors: BOOL;
		(*Reserved Bit 1*)

		(*Reserved Bit 2*)
		(*Reserved Bit 3*)
		(*Reserved Bit 4*)
		(*Reserved Bit 5*)
		(*Reserved Bit 6*)
		(*Reserved Bit 7*)
		(*Reserved Bit 8*)

		Heat2_Data_Exchange_CMD: UINT;
		Heat2_Data_Exchange_CMD_Value: UDINT;



	END_VAR




	(*Set FB_OK to True*)
	FB_OK:= TRUE;

(*$$$$$$$$$$$$$$$$$$$$$$$$$$$$$$$$$$$$$$$$$$$$$$$$Gather Status Of Hardware $$$$$$$$$$$$$$$$$$$$$$$$$$$$$$$$$$$$$$$$$$$$$$$$$$$$*)
	IF NOT External_Terminal_Enable
		THEN (*Internally mapped Profimaster is selected*)
			(*Discrete I/O Node (EL6731 Internal MASTER)*)
			IF Txx_Internal_ProfiMaster.InfoData.State=8
				THEN
				DiscreteNode_OK:=TRUE;
			ELSE
				DiscreteNode_OK:=FALSE;
			END_IF
	END_IF

	IF External_Terminal_Enable
		THEN (*Externally mapped ProfiMaster is selected*)
			(*Discrete I/O Node (EL6731 Internal MASTER)*)
			IF Txx_External_ProfiMaster.InfoData.State=8
				THEN
					DiscreteNode_OK:=TRUE;
			ELSE
					DiscreteNode_OK:=FALSE;
			END_IF
	END_IF

	(*Profibus Node*)
	IF GracoSealer_Inputs.Inputs.DpState=0
		THEN
			ProfiNode_OK:=TRUE;
	ELSE
			ProfiNode_OK:=FALSE;
	END_IF


(*$$$$$$$$$$$$$$$$$$$$$$$$$$$$$$$$$$$$$$$$$$$$$ Gather Safety Inputs $$$$$$$$$$$$$$$$$$$$$$$$$$$$$$$$$$$$$$$$$$$$$$$$$$$$$$$$$*)

(*$$$$$$$$$$$$$$$$$$$$$$$$$$$$$$$$$$$$$$$$$$$$$$$$ Gather Inputs  $$$$$$$$$$$$$$$$$$$$$$$$$$$$$$$$$$$$$$$$$$$$$$$$$$$$*)

(*Graco Sealer Input Bits*)
	Inputs();



(*$$$$$$$$$$$$$$$$$$$$$$$$$$$$$$$$$$$$$$$$$$$$$$$$ Internal Code $$$$$$$$$$$$$$$$$$$$$$$$$$$$$$$$$$$$$$$$$$$$$$$$$$$$$$$$$$$$$$$$$$$$*)





(*$$$$$$$$$$$$$$$$$$$$$$$$$$$$$$$$$$$$$$$$$$$$$$ Transfer Standard Outputs $$$$$$$$$$$$$$$$$$$$$$$$$$$$$$$$$$$$$$$$$$$*)

	(*Output for Dispense Head Amount*)
	Dispense_Amount:= 1;

	(*Bypass Acks*)
	Disp1_Bypass_Ack:= Disp1_Bypass;

	Outputs();























(*end*)

ACTION Inputs:



	(*Pump 1- Inputs from Graco*)
	Pump1_HeartBeat								:= GracoSealer_Inputs.Byte0.0;
	Pump1_Control_Ready							:= GracoSealer_Inputs.Byte0.1;
	Pump1_System_Active							:= GracoSealer_Inputs.Byte0.2;
	Pump1_Control_Active							:= GracoSealer_Inputs.Byte0.3;
	Pump1_NoAlarms_Active						:= GracoSealer_Inputs.Byte0.4;
	Pump1_NoDeviations_Active					:= GracoSealer_Inputs.Byte0.5;
	Pump1_NoAdvisory_Active						:= GracoSealer_Inputs.Byte0.6;
	Pump1_Ready_To_Dispense					:= GracoSealer_Inputs.Byte0.7;


	Pump1_PreCharge_Active						:= GracoSealer_Inputs.Byte1.0;
	Pump1_Dispense_In_Process					:= GracoSealer_Inputs.Byte1.1;
	Pump1_Drum_Low							:= GracoSealer_Inputs.Byte1.2;
	Pump1_Drum_Empty							:= GracoSealer_Inputs.Byte1.3;
	Pump1_Not_Primed							:= GracoSealer_Inputs.Byte1.4;
	Pump1_In_Job_Cycle							:= GracoSealer_Inputs.Byte1.5;
	Pump1_Prime_Active							:= GracoSealer_Inputs.Byte1.6;
	Pump1_Valve_Depressurization_Active			:= GracoSealer_Inputs.Byte1.7;


	Pump1_Platen_Depressurization_Active			:= GracoSealer_Inputs.Byte2.0;
	Pump1_Auto_Depressurization_Active			:= GracoSealer_Inputs.Byte2.1;
	Pump1_Auto_Depressurization_Happened		:= GracoSealer_Inputs.Byte2.2;
	Pump1_Trying_To_Move						:= GracoSealer_Inputs.Byte2.3;
	Pump1_Moving								:= GracoSealer_Inputs.Byte2.4;
	Pump1_DispenseValve_Opened				:= GracoSealer_Inputs.Byte2.5;
	Pump1_PlatenValve_Opened					:= GracoSealer_Inputs.Byte2.6;
	Pump1_Tandem_Active_Pump					:= GracoSealer_Inputs.Byte2.7;			(*0 =Pump 1, 1 = Pump 2*)


	Pump1_EFlo_iQ_Mode_Active					:= GracoSealer_Inputs.Byte3.0;
	Pump1_ChangeOver_Occured					:= GracoSealer_Inputs.Byte3.1;
	(*Reserved Bit 1*)
	(*Reserved Bit 2*)
	(*Reserved Bit 3*)
	(*Reserved Bit 4*)
	(*Reserved Bit 5*)
	(*Reserved Bit 6*)


	Pump1_ActualPump_Flowrate.0					:= GracoSealer_Inputs.Byte4.0;			(*xxxx cc/min*)
	Pump1_ActualPump_Flowrate.1					:= GracoSealer_Inputs.Byte4.1;			(*xxxx cc/min*)
	Pump1_ActualPump_Flowrate.2					:= GracoSealer_Inputs.Byte4.2;			(*xxxx cc/min*)
	Pump1_ActualPump_Flowrate.3					:= GracoSealer_Inputs.Byte4.3;			(*xxxx cc/min*)
	Pump1_ActualPump_Flowrate.4					:= GracoSealer_Inputs.Byte4.4;			(*xxxx cc/min*)
	Pump1_ActualPump_Flowrate.5					:= GracoSealer_Inputs.Byte4.5;			(*xxxx cc/min*)
	Pump1_ActualPump_Flowrate.6					:= GracoSealer_Inputs.Byte4.6;			(*xxxx cc/min*)
	Pump1_ActualPump_Flowrate.7					:= GracoSealer_Inputs.Byte4.7;			(*xxxx cc/min*)

	Pump1_ActualPump_Flowrate.8					:= GracoSealer_Inputs.Byte5.0;			(*xxxx cc/min*)
	Pump1_ActualPump_Flowrate.9					:= GracoSealer_Inputs.Byte5.1;			(*xxxx cc/min*)
	Pump1_ActualPump_Flowrate.10				:= GracoSealer_Inputs.Byte5.2;			(*xxxx cc/min*)
	Pump1_ActualPump_Flowrate.11				:= GracoSealer_Inputs.Byte5.3;			(*xxxx cc/min*)
	Pump1_ActualPump_Flowrate.12				:= GracoSealer_Inputs.Byte5.4;			(*xxxx cc/min*)
	Pump1_ActualPump_Flowrate.13				:= GracoSealer_Inputs.Byte5.5;			(*xxxx cc/min*)
	Pump1_ActualPump_Flowrate.14				:= GracoSealer_Inputs.Byte5.6;			(*xxxx cc/min*)
	Pump1_ActualPump_Flowrate.15				:= GracoSealer_Inputs.Byte5.7;			(*xxxx cc/min*)


	Pump1_Outlet_Pressure.0						:= GracoSealer_Inputs.Byte6.0;			(*xxx.x bar*)
	Pump1_Outlet_Pressure.1						:= GracoSealer_Inputs.Byte6.1;			(*xxx.x bar*)
	Pump1_Outlet_Pressure.2						:= GracoSealer_Inputs.Byte6.2;			(*xxx.x bar*)
	Pump1_Outlet_Pressure.3						:= GracoSealer_Inputs.Byte6.3;			(*xxx.x bar*)
	Pump1_Outlet_Pressure.4						:= GracoSealer_Inputs.Byte6.4;			(*xxx.x bar*)
	Pump1_Outlet_Pressure.5						:= GracoSealer_Inputs.Byte6.5;			(*xxx.x bar*)
	Pump1_Outlet_Pressure.6						:= GracoSealer_Inputs.Byte6.6;			(*xxx.x bar*)
	Pump1_Outlet_Pressure.7						:= GracoSealer_Inputs.Byte6.7;			(*xxx.x bar*)

	Pump1_Outlet_Pressure.8						:= GracoSealer_Inputs.Byte7.0;			(*xxx.x bar*)
	Pump1_Outlet_Pressure.9						:= GracoSealer_Inputs.Byte7.1;			(*xxx.x bar*)
	Pump1_Outlet_Pressure.10						:= GracoSealer_Inputs.Byte7.2;			(*xxx.x bar*)
	Pump1_Outlet_Pressure.11						:= GracoSealer_Inputs.Byte7.3;			(*xxx.x bar*)
	Pump1_Outlet_Pressure.12						:= GracoSealer_Inputs.Byte7.4;			(*xxx.x bar*)
	Pump1_Outlet_Pressure.13						:= GracoSealer_Inputs.Byte7.5;			(*xxx.x bar*)
	Pump1_Outlet_Pressure.14						:= GracoSealer_Inputs.Byte7.6;			(*xxx.x bar*)
	Pump1_Outlet_Pressure.15						:= GracoSealer_Inputs.Byte7.7;			(*xxx.x bar*)


	Pump1_Valve_Pressure.0						:= GracoSealer_Inputs.Byte8.0;			(*xxx.x bar*)
	Pump1_Valve_Pressure.1						:= GracoSealer_Inputs.Byte8.1;			(*xxx.x bar*)
	Pump1_Valve_Pressure.2						:= GracoSealer_Inputs.Byte8.2;			(*xxx.x bar*)
	Pump1_Valve_Pressure.3						:= GracoSealer_Inputs.Byte8.3;			(*xxx.x bar*)
	Pump1_Valve_Pressure.4						:= GracoSealer_Inputs.Byte8.4;			(*xxx.x bar*)
	Pump1_Valve_Pressure.5						:= GracoSealer_Inputs.Byte8.5;			(*xxx.x bar*)
	Pump1_Valve_Pressure.6						:= GracoSealer_Inputs.Byte8.6;			(*xxx.x bar*)
	Pump1_Valve_Pressure.7						:= GracoSealer_Inputs.Byte8.7;			(*xxx.x bar*)

	Pump1_Valve_Pressure.8						:= GracoSealer_Inputs.Byte9.0;			(*xxx.x bar*)
	Pump1_Valve_Pressure.9						:= GracoSealer_Inputs.Byte9.1;			(*xxx.x bar*)
	Pump1_Valve_Pressure.10						:= GracoSealer_Inputs.Byte9.2;			(*xxx.x bar*)
	Pump1_Valve_Pressure.11						:= GracoSealer_Inputs.Byte9.3;			(*xxx.x bar*)
	Pump1_Valve_Pressure.12						:= GracoSealer_Inputs.Byte9.4;			(*xxx.x bar*)
	Pump1_Valve_Pressure.13						:= GracoSealer_Inputs.Byte9.5;			(*xxx.x bar*)
	Pump1_Valve_Pressure.14						:= GracoSealer_Inputs.Byte9.6;			(*xxx.x bar*)
	Pump1_Valve_Pressure.15						:= GracoSealer_Inputs.Byte9.7;			(*xxx.x bar*)


	Pump1_Active_Style_Loaded.0					:= GracoSealer_Inputs.Byte10.0;
	Pump1_Active_Style_Loaded.1					:= GracoSealer_Inputs.Byte10.1;
	Pump1_Active_Style_Loaded.2					:= GracoSealer_Inputs.Byte10.2;
	Pump1_Active_Style_Loaded.3					:= GracoSealer_Inputs.Byte10.3;
	Pump1_Active_Style_Loaded.4					:= GracoSealer_Inputs.Byte10.4;
	Pump1_Active_Style_Loaded.5					:= GracoSealer_Inputs.Byte10.5;
	Pump1_Active_Style_Loaded.6					:= GracoSealer_Inputs.Byte10.6;
	Pump1_Active_Style_Loaded.7					:= GracoSealer_Inputs.Byte10.7;

	Pump1_Active_Style_Loaded.8					:= GracoSealer_Inputs.Byte11.0;
	Pump1_Active_Style_Loaded.9					:= GracoSealer_Inputs.Byte11.1;
	Pump1_Active_Style_Loaded.10					:= GracoSealer_Inputs.Byte11.2;
	Pump1_Active_Style_Loaded.11					:= GracoSealer_Inputs.Byte11.3;
	Pump1_Active_Style_Loaded.12					:= GracoSealer_Inputs.Byte11.4;
	Pump1_Active_Style_Loaded.13					:= GracoSealer_Inputs.Byte11.5;
	Pump1_Active_Style_Loaded.14					:= GracoSealer_Inputs.Byte11.6;
	Pump1_Active_Style_Loaded.15					:= GracoSealer_Inputs.Byte11.7;


	Pump1_Active_Style_Precharge.0				:= GracoSealer_Inputs.Byte12.0; 			(*xxx.x bar*)
	Pump1_Active_Style_Precharge.1				:= GracoSealer_Inputs.Byte12.1; 			(*xxx.x bar*)
	Pump1_Active_Style_Precharge.2				:= GracoSealer_Inputs.Byte12.2; 			(*xxx.x bar*)
	Pump1_Active_Style_Precharge.3				:= GracoSealer_Inputs.Byte12.3; 			(*xxx.x bar*)
	Pump1_Active_Style_Precharge.4				:= GracoSealer_Inputs.Byte12.4; 			(*xxx.x bar*)
	Pump1_Active_Style_Precharge.5				:= GracoSealer_Inputs.Byte12.5; 			(*xxx.x bar*)
	Pump1_Active_Style_Precharge.6				:= GracoSealer_Inputs.Byte12.6; 			(*xxx.x bar*)
	Pump1_Active_Style_Precharge.7				:= GracoSealer_Inputs.Byte12.7; 			(*xxx.x bar*)

	Pump1_Active_Style_Precharge.8				:= GracoSealer_Inputs.Byte13.0; 			(*xxx.x bar*)
	Pump1_Active_Style_Precharge.9				:= GracoSealer_Inputs.Byte13.1; 			(*xxx.x bar*)
	Pump1_Active_Style_Precharge.10				:= GracoSealer_Inputs.Byte13.2; 			(*xxx.x bar*)
	Pump1_Active_Style_Precharge.11				:= GracoSealer_Inputs.Byte13.3; 			(*xxx.x bar*)
	Pump1_Active_Style_Precharge.12				:= GracoSealer_Inputs.Byte13.4; 			(*xxx.x bar*)
	Pump1_Active_Style_Precharge.13				:= GracoSealer_Inputs.Byte13.5; 			(*xxx.x bar*)
	Pump1_Active_Style_Precharge.14				:= GracoSealer_Inputs.Byte13.6; 			(*xxx.x bar*)
	Pump1_Active_Style_Precharge.15				:= GracoSealer_Inputs.Byte13.7; 			(*xxx.x bar*)


	Pump1_Active_Style_Flowrate.0					:= GracoSealer_Inputs.Byte14.0; 	 		(*xxxx cc/min*)
	Pump1_Active_Style_Flowrate.1					:= GracoSealer_Inputs.Byte14.1; 	 		(*xxxx cc/min*)
	Pump1_Active_Style_Flowrate.2					:= GracoSealer_Inputs.Byte14.2; 	 		(*xxxx cc/min*)
	Pump1_Active_Style_Flowrate.3					:= GracoSealer_Inputs.Byte14.3; 	 		(*xxxx cc/min*)
	Pump1_Active_Style_Flowrate.4					:= GracoSealer_Inputs.Byte14.4; 	 		(*xxxx cc/min*)
	Pump1_Active_Style_Flowrate.5					:= GracoSealer_Inputs.Byte14.5; 	 		(*xxxx cc/min*)
	Pump1_Active_Style_Flowrate.6					:= GracoSealer_Inputs.Byte14.6; 	 		(*xxxx cc/min*)
	Pump1_Active_Style_Flowrate.7					:= GracoSealer_Inputs.Byte14.7; 	 		(*xxxx cc/min*)

	Pump1_Active_Style_Flowrate.8					:= GracoSealer_Inputs.Byte15.0; 	 		(*xxxx cc/min*)
	Pump1_Active_Style_Flowrate.9					:= GracoSealer_Inputs.Byte15.1; 	 		(*xxxx cc/min*)
	Pump1_Active_Style_Flowrate.10				:= GracoSealer_Inputs.Byte15.2; 	 		(*xxxx cc/min*)
	Pump1_Active_Style_Flowrate.11				:= GracoSealer_Inputs.Byte15.3; 	 		(*xxxx cc/min*)
	Pump1_Active_Style_Flowrate.12				:= GracoSealer_Inputs.Byte15.4; 	 		(*xxxx cc/min*)
	Pump1_Active_Style_Flowrate.13				:= GracoSealer_Inputs.Byte15.5; 	 		(*xxxx cc/min*)
	Pump1_Active_Style_Flowrate.14				:= GracoSealer_Inputs.Byte15.6; 	 		(*xxxx cc/min*)
	Pump1_Active_Style_Flowrate.15				:= GracoSealer_Inputs.Byte15.7; 	 		(*xxxx cc/min*)


	Pump1_Active_Style_ShotSize.0					:= GracoSealer_Inputs.Byte16.0;  			(*xxx.xx cc*)
	Pump1_Active_Style_ShotSize.1					:= GracoSealer_Inputs.Byte16.1;  			(*xxx.xx cc*)
	Pump1_Active_Style_ShotSize.2					:= GracoSealer_Inputs.Byte16.2;  			(*xxx.xx cc*)
	Pump1_Active_Style_ShotSize.3					:= GracoSealer_Inputs.Byte16.3;  			(*xxx.xx cc*)
	Pump1_Active_Style_ShotSize.4					:= GracoSealer_Inputs.Byte16.4;  			(*xxx.xx cc*)
	Pump1_Active_Style_ShotSize.5					:= GracoSealer_Inputs.Byte16.5;  			(*xxx.xx cc*)
	Pump1_Active_Style_ShotSize.6					:= GracoSealer_Inputs.Byte16.6;  			(*xxx.xx cc*)
	Pump1_Active_Style_ShotSize.7					:= GracoSealer_Inputs.Byte16.7;  			(*xxx.xx cc*)

	Pump1_Active_Style_ShotSize.8					:= GracoSealer_Inputs.Byte17.0;  			(*xxx.xx cc*)
	Pump1_Active_Style_ShotSize.9					:= GracoSealer_Inputs.Byte17.1;  			(*xxx.xx cc*)
	Pump1_Active_Style_ShotSize.10				:= GracoSealer_Inputs.Byte17.2;  			(*xxx.xx cc*)
	Pump1_Active_Style_ShotSize.11				:= GracoSealer_Inputs.Byte17.3;  			(*xxx.xx cc*)
	Pump1_Active_Style_ShotSize.12				:= GracoSealer_Inputs.Byte17.4;  			(*xxx.xx cc*)
	Pump1_Active_Style_ShotSize.13				:= GracoSealer_Inputs.Byte17.5;  			(*xxx.xx cc*)
	Pump1_Active_Style_ShotSize.14				:= GracoSealer_Inputs.Byte17.6;  			(*xxx.xx cc*)
	Pump1_Active_Style_ShotSize.15				:= GracoSealer_Inputs.Byte17.7;  			(*xxx.xx cc*)


	Pump1_Actual_Amount_Dispense.0				:= GracoSealer_Inputs.Byte18.0; 			(*xxxx.xx cc*)
	Pump1_Actual_Amount_Dispense.1				:= GracoSealer_Inputs.Byte18.1; 			(*xxxx.xx cc*)
	Pump1_Actual_Amount_Dispense.2				:= GracoSealer_Inputs.Byte18.2; 			(*xxxx.xx cc*)
	Pump1_Actual_Amount_Dispense.3				:= GracoSealer_Inputs.Byte18.3; 			(*xxxx.xx cc*)
	Pump1_Actual_Amount_Dispense.4				:= GracoSealer_Inputs.Byte18.4; 			(*xxxx.xx cc*)
	Pump1_Actual_Amount_Dispense.5				:= GracoSealer_Inputs.Byte18.5; 			(*xxxx.xx cc*)
	Pump1_Actual_Amount_Dispense.6				:= GracoSealer_Inputs.Byte18.6; 			(*xxxx.xx cc*)
	Pump1_Actual_Amount_Dispense.7				:= GracoSealer_Inputs.Byte18.7; 			(*xxxx.xx cc*)

	Pump1_Actual_Amount_Dispense.8				:= GracoSealer_Inputs.Byte19.0; 			(*xxxx.xx cc*)
	Pump1_Actual_Amount_Dispense.9				:= GracoSealer_Inputs.Byte19.1; 			(*xxxx.xx cc*)
	Pump1_Actual_Amount_Dispense.10				:= GracoSealer_Inputs.Byte19.2; 			(*xxxx.xx cc*)
	Pump1_Actual_Amount_Dispense.11				:= GracoSealer_Inputs.Byte19.3; 			(*xxxx.xx cc*)
	Pump1_Actual_Amount_Dispense.12				:= GracoSealer_Inputs.Byte19.4; 			(*xxxx.xx cc*)
	Pump1_Actual_Amount_Dispense.13				:= GracoSealer_Inputs.Byte19.5; 			(*xxxx.xx cc*)
	Pump1_Actual_Amount_Dispense.14				:= GracoSealer_Inputs.Byte19.6; 			(*xxxx.xx cc*)
	Pump1_Actual_Amount_Dispense.15				:= GracoSealer_Inputs.Byte19.7; 			(*xxxx.xx cc*)

	Pump1_Actual_Amount_Dispense.16				:= GracoSealer_Inputs.Byte20.0; 			(*xxxx.xx cc*)
	Pump1_Actual_Amount_Dispense.17				:= GracoSealer_Inputs.Byte20.1; 			(*xxxx.xx cc*)
	Pump1_Actual_Amount_Dispense.18				:= GracoSealer_Inputs.Byte20.2; 			(*xxxx.xx cc*)
	Pump1_Actual_Amount_Dispense.19				:= GracoSealer_Inputs.Byte20.3; 			(*xxxx.xx cc*)
	Pump1_Actual_Amount_Dispense.20				:= GracoSealer_Inputs.Byte20.4; 			(*xxxx.xx cc*)
	Pump1_Actual_Amount_Dispense.21				:= GracoSealer_Inputs.Byte20.5; 			(*xxxx.xx cc*)
	Pump1_Actual_Amount_Dispense.22				:= GracoSealer_Inputs.Byte20.6; 			(*xxxx.xx cc*)
	Pump1_Actual_Amount_Dispense.23				:= GracoSealer_Inputs.Byte20.7; 			(*xxxx.xx cc*)

	Pump1_Actual_Amount_Dispense.24				:= GracoSealer_Inputs.Byte21.0; 			(*xxxx.xx cc*)
	Pump1_Actual_Amount_Dispense.25				:= GracoSealer_Inputs.Byte21.1; 			(*xxxx.xx cc*)
	Pump1_Actual_Amount_Dispense.26				:= GracoSealer_Inputs.Byte21.2; 			(*xxxx.xx cc*)
	Pump1_Actual_Amount_Dispense.27				:= GracoSealer_Inputs.Byte21.3; 			(*xxxx.xx cc*)
	Pump1_Actual_Amount_Dispense.28				:= GracoSealer_Inputs.Byte21.4; 			(*xxxx.xx cc*)
	Pump1_Actual_Amount_Dispense.29				:= GracoSealer_Inputs.Byte21.5; 			(*xxxx.xx cc*)
	Pump1_Actual_Amount_Dispense.30				:= GracoSealer_Inputs.Byte21.6; 			(*xxxx.xx cc*)
	Pump1_Actual_Amount_Dispense.31				:= GracoSealer_Inputs.Byte21.7; 			(*xxxx.xx cc*)


	Pump1_Actual_Shot_Size.0						:= GracoSealer_Inputs.Byte22.0; 			(*xx.xx cc*)
	Pump1_Actual_Shot_Size.1 						:= GracoSealer_Inputs.Byte22.1; 			(*xx.xx cc*)
	Pump1_Actual_Shot_Size.2						:= GracoSealer_Inputs.Byte22.2; 			(*xx.xx cc*)
	Pump1_Actual_Shot_Size.3						:= GracoSealer_Inputs.Byte22.3; 			(*xx.xx cc*)
	Pump1_Actual_Shot_Size.4						:= GracoSealer_Inputs.Byte22.4; 			(*xx.xx cc*)
	Pump1_Actual_Shot_Size.5						:= GracoSealer_Inputs.Byte22.5; 			(*xx.xx cc*)
	Pump1_Actual_Shot_Size.6						:= GracoSealer_Inputs.Byte22.6; 			(*xx.xx cc*)
	Pump1_Actual_Shot_Size.7						:= GracoSealer_Inputs.Byte22.7; 			(*xx.xx cc*)

	Pump1_Actual_Shot_Size.8						:= GracoSealer_Inputs.Byte23.0; 			(*xx.xx cc*)
	Pump1_Actual_Shot_Size.9						:= GracoSealer_Inputs.Byte23.1; 			(*xx.xx cc*)
	Pump1_Actual_Shot_Size.10					:= GracoSealer_Inputs.Byte23.2; 			(*xx.xx cc*)
	Pump1_Actual_Shot_Size.11					:= GracoSealer_Inputs.Byte23.3; 			(*xx.xx cc*)
	Pump1_Actual_Shot_Size.12					:= GracoSealer_Inputs.Byte23.4; 			(*xx.xx cc*)
	Pump1_Actual_Shot_Size.13					:= GracoSealer_Inputs.Byte23.5; 			(*xx.xx cc*)
	Pump1_Actual_Shot_Size.14					:= GracoSealer_Inputs.Byte23.6; 			(*xx.xx cc*)
	Pump1_Actual_Shot_Size.15					:= GracoSealer_Inputs.Byte23.7; 			(*xx.xx cc*)

	Pump1_Actual_Shot_Size.16					:= GracoSealer_Inputs.Byte24.0; 			(*xx.xx cc*)
	Pump1_Actual_Shot_Size.17					:= GracoSealer_Inputs.Byte24.1; 			(*xx.xx cc*)
	Pump1_Actual_Shot_Size.18					:= GracoSealer_Inputs.Byte24.2; 			(*xx.xx cc*)
	Pump1_Actual_Shot_Size.19					:= GracoSealer_Inputs.Byte24.3; 			(*xx.xx cc*)
	Pump1_Actual_Shot_Size.20					:= GracoSealer_Inputs.Byte24.4; 			(*xx.xx cc*)
	Pump1_Actual_Shot_Size.21					:= GracoSealer_Inputs.Byte24.5; 			(*xx.xx cc*)
	Pump1_Actual_Shot_Size.22					:= GracoSealer_Inputs.Byte24.6; 			(*xx.xx cc*)
	Pump1_Actual_Shot_Size.23					:= GracoSealer_Inputs.Byte24.7; 			(*xx.xx cc*)

	Pump1_Actual_Shot_Size.24					:= GracoSealer_Inputs.Byte25.0; 			(*xx.xx cc*)
	Pump1_Actual_Shot_Size.25					:= GracoSealer_Inputs.Byte25.1; 			(*xx.xx cc*)
	Pump1_Actual_Shot_Size.26					:= GracoSealer_Inputs.Byte25.2; 			(*xx.xx cc*)
	Pump1_Actual_Shot_Size.27					:= GracoSealer_Inputs.Byte25.3; 			(*xx.xx cc*)
	Pump1_Actual_Shot_Size.28					:= GracoSealer_Inputs.Byte25.4; 			(*xx.xx cc*)
	Pump1_Actual_Shot_Size.29					:= GracoSealer_Inputs.Byte25.5; 			(*xx.xx cc*)
	Pump1_Actual_Shot_Size.30					:= GracoSealer_Inputs.Byte25.6; 			(*xx.xx cc*)
	Pump1_Actual_Shot_Size.31					:= GracoSealer_Inputs.Byte25.7; 			(*xx.xx cc*)


	Pump1_Actual_Style_PreCharge_REQ.0			:= GracoSealer_Inputs.Byte26.0;			(*xxx.x bar*)
	Pump1_Actual_Style_PreCharge_REQ.1			:= GracoSealer_Inputs.Byte26.1;			(*xxx.x bar*)
	Pump1_Actual_Style_PreCharge_REQ.2			:= GracoSealer_Inputs.Byte26.2;			(*xxx.x bar*)
	Pump1_Actual_Style_PreCharge_REQ.3			:= GracoSealer_Inputs.Byte26.3;			(*xxx.x bar*)
	Pump1_Actual_Style_PreCharge_REQ.4			:= GracoSealer_Inputs.Byte26.4;			(*xxx.x bar*)
	Pump1_Actual_Style_PreCharge_REQ.5			:= GracoSealer_Inputs.Byte26.5;			(*xxx.x bar*)
	Pump1_Actual_Style_PreCharge_REQ.6			:= GracoSealer_Inputs.Byte26.6;			(*xxx.x bar*)
	Pump1_Actual_Style_PreCharge_REQ.7			:= GracoSealer_Inputs.Byte26.7;			(*xxx.x bar*)

	Pump1_Actual_Style_PreCharge_REQ.8			:= GracoSealer_Inputs.Byte27.0;			(*xxx.x bar*)
	Pump1_Actual_Style_PreCharge_REQ.9			:= GracoSealer_Inputs.Byte27.1;			(*xxx.x bar*)
	Pump1_Actual_Style_PreCharge_REQ.10			:= GracoSealer_Inputs.Byte27.2;			(*xxx.x bar*)
	Pump1_Actual_Style_PreCharge_REQ.11			:= GracoSealer_Inputs.Byte27.3;			(*xxx.x bar*)
	Pump1_Actual_Style_PreCharge_REQ.12			:= GracoSealer_Inputs.Byte27.4;			(*xxx.x bar*)
	Pump1_Actual_Style_PreCharge_REQ.13			:= GracoSealer_Inputs.Byte27.5;			(*xxx.x bar*)
	Pump1_Actual_Style_PreCharge_REQ.14			:= GracoSealer_Inputs.Byte27.6;			(*xxx.x bar*)
	Pump1_Actual_Style_PreCharge_REQ.15			:= GracoSealer_Inputs.Byte27.7;			(*xxx.x bar*)


	Pump1_Actual_Style_Flowrate_REQ.0			:= GracoSealer_Inputs.Byte28.0;			(*xxxx cc/min*)
	Pump1_Actual_Style_Flowrate_REQ.1			:= GracoSealer_Inputs.Byte28.1;			(*xxxx cc/min*)
	Pump1_Actual_Style_Flowrate_REQ.2			:= GracoSealer_Inputs.Byte28.2;			(*xxxx cc/min*)
	Pump1_Actual_Style_Flowrate_REQ.3			:= GracoSealer_Inputs.Byte28.3;			(*xxxx cc/min*)
	Pump1_Actual_Style_Flowrate_REQ.4			:= GracoSealer_Inputs.Byte28.4;			(*xxxx cc/min*)
	Pump1_Actual_Style_Flowrate_REQ.5			:= GracoSealer_Inputs.Byte28.5;			(*xxxx cc/min*)
	Pump1_Actual_Style_Flowrate_REQ.6			:= GracoSealer_Inputs.Byte28.6;			(*xxxx cc/min*)
	Pump1_Actual_Style_Flowrate_REQ.7			:= GracoSealer_Inputs.Byte28.7;			(*xxxx cc/min*)

	Pump1_Actual_Style_Flowrate_REQ.8			:= GracoSealer_Inputs.Byte29.0;			(*xxxx cc/min*)
	Pump1_Actual_Style_Flowrate_REQ.9			:= GracoSealer_Inputs.Byte29.1;			(*xxxx cc/min*)
	Pump1_Actual_Style_Flowrate_REQ.10			:= GracoSealer_Inputs.Byte29.2;			(*xxxx cc/min*)
	Pump1_Actual_Style_Flowrate_REQ.11			:= GracoSealer_Inputs.Byte29.3;			(*xxxx cc/min*)
	Pump1_Actual_Style_Flowrate_REQ.12			:= GracoSealer_Inputs.Byte29.4;			(*xxxx cc/min*)
	Pump1_Actual_Style_Flowrate_REQ.13			:= GracoSealer_Inputs.Byte29.5;			(*xxxx cc/min*)
	Pump1_Actual_Style_Flowrate_REQ.14			:= GracoSealer_Inputs.Byte29.6;			(*xxxx cc/min*)
	Pump1_Actual_Style_Flowrate_REQ.15			:= GracoSealer_Inputs.Byte29.7;			(*xxxx cc/min*)


	Pump1_Actual_Style_Shot_Size_REQ.0			:= GracoSealer_Inputs.Byte30.0;			(*xxx.xx cc*)
	Pump1_Actual_Style_Shot_Size_REQ.1			:= GracoSealer_Inputs.Byte30.1;			(*xxx.xx cc*)
	Pump1_Actual_Style_Shot_Size_REQ.2			:= GracoSealer_Inputs.Byte30.2;			(*xxx.xx cc*)
	Pump1_Actual_Style_Shot_Size_REQ.3			:= GracoSealer_Inputs.Byte30.3;			(*xxx.xx cc*)
	Pump1_Actual_Style_Shot_Size_REQ.4			:= GracoSealer_Inputs.Byte30.4;			(*xxx.xx cc*)
	Pump1_Actual_Style_Shot_Size_REQ.5			:= GracoSealer_Inputs.Byte30.5;			(*xxx.xx cc*)
	Pump1_Actual_Style_Shot_Size_REQ.6			:= GracoSealer_Inputs.Byte30.6;			(*xxx.xx cc*)
	Pump1_Actual_Style_Shot_Size_REQ.7			:= GracoSealer_Inputs.Byte30.7;			(*xxx.xx cc*)

	Pump1_Actual_Style_Shot_Size_REQ.8			:= GracoSealer_Inputs.Byte31.0;			(*xxx.xx cc*)
	Pump1_Actual_Style_Shot_Size_REQ.9			:= GracoSealer_Inputs.Byte31.1;			(*xxx.xx cc*)
	Pump1_Actual_Style_Shot_Size_REQ.10			:= GracoSealer_Inputs.Byte31.2;			(*xxx.xx cc*)
	Pump1_Actual_Style_Shot_Size_REQ.11			:= GracoSealer_Inputs.Byte31.3;			(*xxx.xx cc*)
	Pump1_Actual_Style_Shot_Size_REQ.12			:= GracoSealer_Inputs.Byte31.4;			(*xxx.xx cc*)
	Pump1_Actual_Style_Shot_Size_REQ.13			:= GracoSealer_Inputs.Byte31.5;			(*xxx.xx cc*)
	Pump1_Actual_Style_Shot_Size_REQ.14			:= GracoSealer_Inputs.Byte31.6;			(*xxx.xx cc*)
	Pump1_Actual_Style_Shot_Size_REQ.15			:= GracoSealer_Inputs.Byte31.7;			(*xxx.xx cc*)


	Pump1_PumpPosition.0						:= GracoSealer_Inputs.Byte32.0;			(*x.xxxx inches*)
	Pump1_PumpPosition.1						:= GracoSealer_Inputs.Byte32.1;			(*x.xxxx inches*)
	Pump1_PumpPosition.2						:= GracoSealer_Inputs.Byte32.2;			(*x.xxxx inches*)
	Pump1_PumpPosition.3						:= GracoSealer_Inputs.Byte32.3;			(*x.xxxx inches*)
	Pump1_PumpPosition.4						:= GracoSealer_Inputs.Byte32.4;			(*x.xxxx inches*)
	Pump1_PumpPosition.5						:= GracoSealer_Inputs.Byte32.5;			(*x.xxxx inches*)
	Pump1_PumpPosition.6						:= GracoSealer_Inputs.Byte32.6;			(*x.xxxx inches*)
	Pump1_PumpPosition.7						:= GracoSealer_Inputs.Byte32.7;			(*x.xxxx inches*)

	Pump1_PumpPosition.8						:= GracoSealer_Inputs.Byte33.0;			(*x.xxxx inches*)
	Pump1_PumpPosition.9						:= GracoSealer_Inputs.Byte33.1;			(*x.xxxx inches*)
	Pump1_PumpPosition.10						:= GracoSealer_Inputs.Byte33.2;			(*x.xxxx inches*)
	Pump1_PumpPosition.11						:= GracoSealer_Inputs.Byte33.3;			(*x.xxxx inches*)
	Pump1_PumpPosition.12						:= GracoSealer_Inputs.Byte33.4;			(*x.xxxx inches*)
	Pump1_PumpPosition.13						:= GracoSealer_Inputs.Byte33.5;			(*x.xxxx inches*)
	Pump1_PumpPosition.14						:= GracoSealer_Inputs.Byte33.6;			(*x.xxxx inches*)
	Pump1_PumpPosition.15						:= GracoSealer_Inputs.Byte33.7;			(*x.xxxx inches*)


	Pump1_Data_Exchange_Active_CMD.0			:= GracoSealer_Inputs.Byte34.0;
	Pump1_Data_Exchange_Active_CMD.1			:= GracoSealer_Inputs.Byte34.1;
	Pump1_Data_Exchange_Active_CMD.2			:= GracoSealer_Inputs.Byte34.2;
	Pump1_Data_Exchange_Active_CMD.3			:= GracoSealer_Inputs.Byte34.3;
	Pump1_Data_Exchange_Active_CMD.4			:= GracoSealer_Inputs.Byte34.4;
	Pump1_Data_Exchange_Active_CMD.5			:= GracoSealer_Inputs.Byte34.5;
	Pump1_Data_Exchange_Active_CMD.6			:= GracoSealer_Inputs.Byte34.6;
	Pump1_Data_Exchange_Active_CMD.7			:= GracoSealer_Inputs.Byte34.7;

	Pump1_Data_Exchange_Active_CMD.8			:= GracoSealer_Inputs.Byte35.0;
	Pump1_Data_Exchange_Active_CMD.9			:= GracoSealer_Inputs.Byte35.1;
	Pump1_Data_Exchange_Active_CMD.10			:= GracoSealer_Inputs.Byte35.2;
	Pump1_Data_Exchange_Active_CMD.11			:= GracoSealer_Inputs.Byte35.3;
	Pump1_Data_Exchange_Active_CMD.12			:= GracoSealer_Inputs.Byte35.4;
	Pump1_Data_Exchange_Active_CMD.13			:= GracoSealer_Inputs.Byte35.5;
	Pump1_Data_Exchange_Active_CMD.14			:= GracoSealer_Inputs.Byte35.6;
	Pump1_Data_Exchange_Active_CMD.15			:= GracoSealer_Inputs.Byte35.7;


	Pump1_Data_Exchange_Active_CMD_Value.0		:= GracoSealer_Inputs.Byte36.0;
	Pump1_Data_Exchange_Active_CMD_Value.1		:= GracoSealer_Inputs.Byte36.1;
	Pump1_Data_Exchange_Active_CMD_Value.2		:= GracoSealer_Inputs.Byte36.2;
	Pump1_Data_Exchange_Active_CMD_Value.3		:= GracoSealer_Inputs.Byte36.3;
	Pump1_Data_Exchange_Active_CMD_Value.4		:= GracoSealer_Inputs.Byte36.4;
	Pump1_Data_Exchange_Active_CMD_Value.5		:= GracoSealer_Inputs.Byte36.5;
	Pump1_Data_Exchange_Active_CMD_Value.6		:= GracoSealer_Inputs.Byte36.6;
	Pump1_Data_Exchange_Active_CMD_Value.7		:= GracoSealer_Inputs.Byte36.7;

	Pump1_Data_Exchange_Active_CMD_Value.8		:= GracoSealer_Inputs.Byte37.0;
	Pump1_Data_Exchange_Active_CMD_Value.9		:= GracoSealer_Inputs.Byte37.1;
	Pump1_Data_Exchange_Active_CMD_Value.10	:= GracoSealer_Inputs.Byte37.2;
	Pump1_Data_Exchange_Active_CMD_Value.11	:= GracoSealer_Inputs.Byte37.3;
	Pump1_Data_Exchange_Active_CMD_Value.12	:= GracoSealer_Inputs.Byte37.4;
	Pump1_Data_Exchange_Active_CMD_Value.13	:= GracoSealer_Inputs.Byte37.5;
	Pump1_Data_Exchange_Active_CMD_Value.14	:= GracoSealer_Inputs.Byte37.6;
	Pump1_Data_Exchange_Active_CMD_Value.15	:= GracoSealer_Inputs.Byte37.7;
	Pump1_Data_Exchange_Active_CMD_Value.16	:= GracoSealer_Inputs.Byte38.0;
	Pump1_Data_Exchange_Active_CMD_Value.17	:= GracoSealer_Inputs.Byte38.1;
	Pump1_Data_Exchange_Active_CMD_Value.18	:= GracoSealer_Inputs.Byte38.2;
	Pump1_Data_Exchange_Active_CMD_Value.19	:= GracoSealer_Inputs.Byte38.3;
	Pump1_Data_Exchange_Active_CMD_Value.20	:= GracoSealer_Inputs.Byte38.4;
	Pump1_Data_Exchange_Active_CMD_Value.21	:= GracoSealer_Inputs.Byte38.5;
	Pump1_Data_Exchange_Active_CMD_Value.22	:= GracoSealer_Inputs.Byte38.6;
	Pump1_Data_Exchange_Active_CMD_Value.23	:= GracoSealer_Inputs.Byte38.7;

	Pump1_Data_Exchange_Active_CMD_Value.24	:= GracoSealer_Inputs.Byte39.0;
	Pump1_Data_Exchange_Active_CMD_Value.25	:= GracoSealer_Inputs.Byte39.1;
	Pump1_Data_Exchange_Active_CMD_Value.26	:= GracoSealer_Inputs.Byte39.2;
	Pump1_Data_Exchange_Active_CMD_Value.27	:= GracoSealer_Inputs.Byte39.3;
	Pump1_Data_Exchange_Active_CMD_Value.28	:= GracoSealer_Inputs.Byte39.4;
	Pump1_Data_Exchange_Active_CMD_Value.29	:= GracoSealer_Inputs.Byte39.5;
	Pump1_Data_Exchange_Active_CMD_Value.30	:= GracoSealer_Inputs.Byte39.6;
	Pump1_Data_Exchange_Active_CMD_Value.31	:= GracoSealer_Inputs.Byte39.7;



	(*Pump 2 - Inputs Only used for Tandem systems*)
	Pump2_HeartBeat								:= GracoSealer_Inputs.Byte40.0;
	Pump2_Control_Ready							:= GracoSealer_Inputs.Byte40.1;
	Pump2_System_Active							:= GracoSealer_Inputs.Byte40.2;
	Pump2_Control_Active							:= GracoSealer_Inputs.Byte40.3;
	Pump2_NoAlarms_Active						:= GracoSealer_Inputs.Byte40.4;
	Pump2_NoDeviations_Active					:= GracoSealer_Inputs.Byte40.5;
	Pump2_NoAdvisory_Active						:= GracoSealer_Inputs.Byte40.6;
	Pump2_Ready_To_Dispense					:= GracoSealer_Inputs.Byte40.7;


	Pump2_PreCharge_Active						:= GracoSealer_Inputs.Byte41.0;
	Pump2_Dispense_In_Process					:= GracoSealer_Inputs.Byte41.1;
	Pump2_Drum_Low							:= GracoSealer_Inputs.Byte41.2;
	Pump2_Drum_Empty							:= GracoSealer_Inputs.Byte41.3;
	Pump2_Not_Primed							:= GracoSealer_Inputs.Byte41.4;
	Pump2_In_Job_Cycle							:= GracoSealer_Inputs.Byte41.5;
	Pump2_Prime_Active							:= GracoSealer_Inputs.Byte41.6;
	Pump2_Valve_Depressurization_Active			:= GracoSealer_Inputs.Byte41.7;


	Pump2_Platen_Depressurization_Active			:= GracoSealer_Inputs.Byte42.0;
	Pump2_Auto_Depressurization_Active			:= GracoSealer_Inputs.Byte42.1;
	Pump2_Auto_Depressurization_Happened		:= GracoSealer_Inputs.Byte42.2;
	Pump2_Trying_To_Move						:= GracoSealer_Inputs.Byte42.3;
	Pump2_Moving								:= GracoSealer_Inputs.Byte42.4;
	Pump2_DispenseValve_Opened				:= GracoSealer_Inputs.Byte42.5;
	Pump2_PlatenValve_Opened					:= GracoSealer_Inputs.Byte42.6;
	Pump2_Tandem_Active_Pump					:= GracoSealer_Inputs.Byte42.7;			(*0 =Pump 1, 1 = Pump 2*)


	Pump2_EFlo_iQ_Mode_Active					:= GracoSealer_Inputs.Byte43.0;
	(*Reserved Bit 1*)
	(*Reserved Bit 2*)
	(*Reserved Bit 3*)
	(*Reserved Bit 4*)
	(*Reserved Bit 5*)
	(*Reserved Bit 6*)
	(*Reserved Bit 7*)
	(*Reserved Bit 8*)
	(*Reserved Bit 9*)


	Pump2_ActualPump_Flowrate.0					:= GracoSealer_Inputs.Byte44.0;			(*xxxx cc/min*)
	Pump2_ActualPump_Flowrate.1					:= GracoSealer_Inputs.Byte44.1;			(*xxxx cc/min*)
	Pump2_ActualPump_Flowrate.2					:= GracoSealer_Inputs.Byte44.2;			(*xxxx cc/min*)
	Pump2_ActualPump_Flowrate.3					:= GracoSealer_Inputs.Byte44.3;			(*xxxx cc/min*)
	Pump2_ActualPump_Flowrate.4					:= GracoSealer_Inputs.Byte44.4;			(*xxxx cc/min*)
	Pump2_ActualPump_Flowrate.5					:= GracoSealer_Inputs.Byte44.5;			(*xxxx cc/min*)
	Pump2_ActualPump_Flowrate.6					:= GracoSealer_Inputs.Byte44.6;			(*xxxx cc/min*)
	Pump2_ActualPump_Flowrate.7					:= GracoSealer_Inputs.Byte44.7;			(*xxxx cc/min*)

	Pump2_ActualPump_Flowrate.8					:= GracoSealer_Inputs.Byte45.0;			(*xxxx cc/min*)
	Pump2_ActualPump_Flowrate.9					:= GracoSealer_Inputs.Byte45.1;			(*xxxx cc/min*)
	Pump2_ActualPump_Flowrate.10				:= GracoSealer_Inputs.Byte45.2;			(*xxxx cc/min*)
	Pump2_ActualPump_Flowrate.11				:= GracoSealer_Inputs.Byte45.3;			(*xxxx cc/min*)
	Pump2_ActualPump_Flowrate.12				:= GracoSealer_Inputs.Byte45.4;			(*xxxx cc/min*)
	Pump2_ActualPump_Flowrate.13				:= GracoSealer_Inputs.Byte45.5;			(*xxxx cc/min*)
	Pump2_ActualPump_Flowrate.14				:= GracoSealer_Inputs.Byte45.6;			(*xxxx cc/min*)
	Pump2_ActualPump_Flowrate.15				:= GracoSealer_Inputs.Byte45.7;			(*xxxx cc/min*)


	Pump2_Outlet_Pressure.0						:= GracoSealer_Inputs.Byte46.0;			(*xxx.x bar*)
	Pump2_Outlet_Pressure.1						:= GracoSealer_Inputs.Byte46.1;			(*xxx.x bar*)
	Pump2_Outlet_Pressure.2						:= GracoSealer_Inputs.Byte46.2;			(*xxx.x bar*)
	Pump2_Outlet_Pressure.3						:= GracoSealer_Inputs.Byte46.3;			(*xxx.x bar*)
	Pump2_Outlet_Pressure.4						:= GracoSealer_Inputs.Byte46.4;			(*xxx.x bar*)
	Pump2_Outlet_Pressure.5						:= GracoSealer_Inputs.Byte46.5;			(*xxx.x bar*)
	Pump2_Outlet_Pressure.6						:= GracoSealer_Inputs.Byte46.6;			(*xxx.x bar*)
	Pump2_Outlet_Pressure.7						:= GracoSealer_Inputs.Byte46.7;			(*xxx.x bar*)

	Pump2_Outlet_Pressure.8						:= GracoSealer_Inputs.Byte47.0;			(*xxx.x bar*)
	Pump2_Outlet_Pressure.9						:= GracoSealer_Inputs.Byte47.1;			(*xxx.x bar*)
	Pump2_Outlet_Pressure.10						:= GracoSealer_Inputs.Byte47.2;			(*xxx.x bar*)
	Pump2_Outlet_Pressure.11						:= GracoSealer_Inputs.Byte47.3;			(*xxx.x bar*)
	Pump2_Outlet_Pressure.12						:= GracoSealer_Inputs.Byte47.4;			(*xxx.x bar*)
	Pump2_Outlet_Pressure.13						:= GracoSealer_Inputs.Byte47.5;			(*xxx.x bar*)
	Pump2_Outlet_Pressure.14						:= GracoSealer_Inputs.Byte47.6;			(*xxx.x bar*)
	Pump2_Outlet_Pressure.15						:= GracoSealer_Inputs.Byte47.7;			(*xxx.x bar*)


	Pump2_Data_Exchange_Active_CMD.0			:= GracoSealer_Inputs.Byte48.0;
	Pump2_Data_Exchange_Active_CMD.1			:= GracoSealer_Inputs.Byte48.1;
	Pump2_Data_Exchange_Active_CMD.2			:= GracoSealer_Inputs.Byte48.2;
	Pump2_Data_Exchange_Active_CMD.3			:= GracoSealer_Inputs.Byte48.3;
	Pump2_Data_Exchange_Active_CMD.4			:= GracoSealer_Inputs.Byte48.4;
	Pump2_Data_Exchange_Active_CMD.5			:= GracoSealer_Inputs.Byte48.5;
	Pump2_Data_Exchange_Active_CMD.6			:= GracoSealer_Inputs.Byte48.6;
	Pump2_Data_Exchange_Active_CMD.7			:= GracoSealer_Inputs.Byte48.7;

	Pump2_Data_Exchange_Active_CMD.8			:= GracoSealer_Inputs.Byte49.0;
	Pump2_Data_Exchange_Active_CMD.9			:= GracoSealer_Inputs.Byte49.1;
	Pump2_Data_Exchange_Active_CMD.10			:= GracoSealer_Inputs.Byte49.2;
	Pump2_Data_Exchange_Active_CMD.11			:= GracoSealer_Inputs.Byte49.3;
	Pump2_Data_Exchange_Active_CMD.12			:= GracoSealer_Inputs.Byte49.4;
	Pump2_Data_Exchange_Active_CMD.13			:= GracoSealer_Inputs.Byte49.5;
	Pump2_Data_Exchange_Active_CMD.14			:= GracoSealer_Inputs.Byte49.6;
	Pump2_Data_Exchange_Active_CMD.15			:= GracoSealer_Inputs.Byte49.7;


	Pump2_Data_Exchange_Active_CMD_Value.0		:= GracoSealer_Inputs.Byte50.0;
	Pump2_Data_Exchange_Active_CMD_Value.1		:= GracoSealer_Inputs.Byte50.1;
	Pump2_Data_Exchange_Active_CMD_Value.2		:= GracoSealer_Inputs.Byte50.2;
	Pump2_Data_Exchange_Active_CMD_Value.3		:= GracoSealer_Inputs.Byte50.3;
	Pump2_Data_Exchange_Active_CMD_Value.4		:= GracoSealer_Inputs.Byte50.4;
	Pump2_Data_Exchange_Active_CMD_Value.5		:= GracoSealer_Inputs.Byte50.5;
	Pump2_Data_Exchange_Active_CMD_Value.6		:= GracoSealer_Inputs.Byte50.6;
	Pump2_Data_Exchange_Active_CMD_Value.7		:= GracoSealer_Inputs.Byte50.7;

	Pump2_Data_Exchange_Active_CMD_Value.8		:= GracoSealer_Inputs.Byte51.0;
	Pump2_Data_Exchange_Active_CMD_Value.9		:= GracoSealer_Inputs.Byte51.1;
	Pump2_Data_Exchange_Active_CMD_Value.10	:= GracoSealer_Inputs.Byte51.2;
	Pump2_Data_Exchange_Active_CMD_Value.11	:= GracoSealer_Inputs.Byte51.3;
	Pump2_Data_Exchange_Active_CMD_Value.12	:= GracoSealer_Inputs.Byte51.4;
	Pump2_Data_Exchange_Active_CMD_Value.13	:= GracoSealer_Inputs.Byte51.5;
	Pump2_Data_Exchange_Active_CMD_Value.14	:= GracoSealer_Inputs.Byte51.6;
	Pump2_Data_Exchange_Active_CMD_Value.15	:= GracoSealer_Inputs.Byte51.7;

